(* POU _FB_BACnet_AdsConn, ST *)
FUNCTION_BLOCK _FB_BACnet_AdsConn
VAR_INPUT
	bAutoReload			: BOOL := TRUE; (* TRUE --> reload on device operational state and other changes *)
	bReload				: BOOL; (* FALSE --> TRUE refresh information *)
	bIsClient			: BOOL; (* TRUE --> Connection with client device (remote server) *)
END_VAR
VAR_IN_OUT
	bDevOperational		: BOOL;
	sAmsNetId			: T_AmsNetId;
	tDevObjId			: T_BACnet_ObjectIdentifier;
END_VAR
VAR_OUTPUT
	bReady				: BOOL;
	bBusy				: BOOL;
	bDone				: BOOL;
	bError				: BOOL;
	nErrorId			: UINT;
	stBACnetAds			: ST_BACnet_AdsConnection;
END_VAR
VAR
	_BACnetAmsNetID		: T_AmsNetId;
	_fbAdsRead			: FW_AdsRead;
	_arrAdsBuf			: ARRAY[0..13] OF DWORD;
	_rtrigReload		: R_TRIG;
	_rtrigOP			: R_TRIG;
	_i					: INT;
	_nDevObjects		: UDINT;
	_nObjIdx			: UDINT;
	_nAmsPort			: UINT;
	_tObjId				: T_BACnet_ObjectIdentifier := 16#FFFFFFFF;
END_VAR
(*
#define ADSIGRP_BACNET_CLIENT_COM_PARAMETER                      0x010

typedef struct _BACnetDevComData
{
      BACnetObjectIdentifier deviceObjIdentifier;
      BACnetAddress                  netAddress;                      // 10 Byte
      WORD                                 UdpPort;
      DWORD                                IPadress;       
      WORD                                 maxApdu;                         // wird im "Iam" Frame gesetzt
      WORD                                 vendorId;                        // wird im "Iam" Frame gesetzt
      DWORD                                maxSegments;                     // 0 == unspecified number of segments
      DWORD                                segmentTimeout;            // wenn 0 dann Defaultwerte des Devices nehmen 
      DWORD                                apduTimeout;                     // wenn 0 dann Defaultwerte des Devices nehmen
      DWORD                                nApduRetries;              // wenn 0 dann Defaultwerte des Devices nehmen
      BYTE                                 ethernetMacAddr[6];   // Ethernet MAC Address
      BYTE                                 segmentsSupported;         // segmentation both, transmit, receive, no (0 == segmentation both)
      BYTE                                 reserved;
} BACnetDevComData, *PBACnetDevComData;

-----------------------------------------------------
Server:

AdsReadInd, IndexGroup:
#define ADSIGRP_BACNET_GET_OBJECT_LIST                                 0x009

indexOffset == 0 -> Anzahl der Objekte

gerader Index -> Objekttyp
ungerader Index -> ObjetInstanz

IndexOffset 2 sollte daher die DeviceID des Servers sein
*)

(* ads communication *)
_fbAdsRead(
	sNetId		:= _BACnetAmsNetID,
	nPort		:= ,
	nIdxGrp		:= ,
	nIdxOffs	:= ,
	cbReadLen	:= SIZEOF(_arrAdsBuf),
	pReadBuff	:= ADR(_arrAdsBuf),
	bExecute	:= ,
	tTimeout	:= BACnet_ADSTimeOut,
	bBusy		=> ,
	bError		=> ,
	nErrId		=> ,
	cbRead		=> );

(* catch reload event trigger *)
_rtrigReload(CLK:= bReload, Q=> );
_rtrigOP(CLK:= bDevOperational, Q=> );

(* state machine *)
CASE _i OF

	0: (* Idle *)
		IF sAmsNetId = '' THEN
			(* NetId not OK, return with error *)
			nErrorId := BACnet_ERR_ADS_NO_VALID_NET_ID;
			stBACnetAds.bValid := FALSE;
			_BACnetAmsNetID := '';
		ELSIF (F_BACnet_GetObjType(tDevObjId) <> BACnetObjectType_Device) THEN
			(* Object type is not device *)
			nErrorId := BACnet_ERR_ADS_ObjectId;
			stBACnetAds.bValid := FALSE;
			_tObjId := 0;
		ELSIF	_rtrigReload.Q
			OR	(		(		(sAmsNetId <> stBACnetAds.sAmsNetId)
							OR	(tDevObjId <> _tObjId)
							OR	(_BACnetAmsNetID <> sAmsNetId)
							OR	_rtrigOP.Q
						)
					AND	bAutoReload
				)
		THEN
			IF (NOT bDevOperational) THEN
				(* BACnet adapter error *)
				nErrorId := BACnet_ERR_ADS_DeviceOP;
				stBACnetAds.bValid := FALSE;
			ELSE
				nErrorId := BACnet_ERR_NO_ERROR;
				_i := 1;
				(* store connection info *)
				_BACnetAmsNetID	:= sAmsNetId;
				_tObjId := tDevObjId;
			END_IF
		END_IF
		bDone := FALSE;

	(* Determin the AMS port *)
	1:
		IF _fbAdsRead.bExecute THEN
			IF _fbAdsRead.bError THEN
				IF ((UDINT_TO_DWORD(_fbAdsRead.nErrId) AND 16#0000FFFF) = 16#0703) THEN
					(* couldn't read service for AMS port of the device - maybe R6 stack running *)
					nErrorId := BACnet_ERR_ADS_LegacyStack;
				ELSE
					nErrorId := BACnet_ERR_ADS_Read;
				END_IF
				_fbAdsRead.bExecute := FALSE;
				_i := 100;
				stBACnetAds.bValid := FALSE;
			ELSIF (NOT _fbAdsRead.bBusy) THEN
				_fbAdsRead.bExecute := FALSE;
				(* check if port info is valid *)
				IF (_fbAdsRead.cbRead = 2) THEN
					_nAmsPort := DWORD_TO_UINT(_arrAdsBuf[0] AND 16#0000FFFF);
					(* length ok? *)
					IF _nAmsPort >= 1000 THEN
						IF bIsClient THEN
							_i := 100;
							stBACnetAds.nDeviceId := F_BACnet_GetObjInstance(tDevObjId);
						ELSE
							_i := 11;
						END_IF
					ELSE
						(* wrong length, abort *)
						_i := 100;
						nErrorId := BACnet_ERR_ADS_AmsPort;
						stBACnetAds.bValid := FALSE;
					END_IF
				ELSE
					nErrorId := BACnet_ERR_ADS_Data;
					_i := 100;
					stBACnetAds.bValid := FALSE;
				END_IF
			END_IF
		ELSE
			(* start ADS reading *)
			_fbAdsRead.bExecute := TRUE;
			_fbAdsRead.nIdxGrp := BACnet_ADSIGRP_DEV_R_GETADSPORTBYDEVID;
			_fbAdsRead.nPort := 65535;
			_fbAdsRead.nIdxOffs := tDevObjId;
		END_IF

	(* try READ server info -object list length- *)
	11:
		IF _fbAdsRead.bExecute THEN
			IF _fbAdsRead.bError THEN
				_fbAdsRead.bExecute := FALSE;
				_i := 100;
				nErrorId := BACnet_ERR_ADS_Read;
				stBACnetAds.bValid := FALSE;
			ELSIF (NOT _fbAdsRead.bBusy) THEN
				_fbAdsRead.bExecute := FALSE;
				(* check if object list is valid *)
				IF (_fbAdsRead.cbRead = 4) THEN
					_nDevObjects := _arrAdsBuf[0];
					(* length ok? *)
					IF _nDevObjects >= 1 THEN
						_i := 12;
						_nObjIdx := 0;
					ELSE
						(* wrong length, abort *)
						_i := 100;
						nErrorId := BACnet_ERR_ADS_ObjListEmpty;
						stBACnetAds.bValid := FALSE;
					END_IF
				ELSE
					nErrorId := BACnet_ERR_ADS_Data;
					_i := 100;
					stBACnetAds.bValid := FALSE;
				END_IF
			END_IF
		ELSE
			(* start ADS reading *)
			_fbAdsRead.bExecute := TRUE;
			_fbAdsRead.nIdxGrp := BACnet_ADSIGRP_GET_OBJECT_LIST;
			_fbAdsRead.nPort := _nAmsPort;
			_fbAdsRead.nIdxOffs := 0;
		END_IF

	(* try READ server info -object type- *)
	12:
		IF _fbAdsRead.bExecute THEN
			IF _fbAdsRead.bError THEN
				_fbAdsRead.bExecute := FALSE;
				_i := 100;
				nErrorId := BACnet_ERR_ADS_Read;
				stBACnetAds.bValid := FALSE;
			ELSIF (NOT _fbAdsRead.bBusy) THEN
				_fbAdsRead.bExecute := FALSE;
				(* check if type is valid *)
				IF (_fbAdsRead.cbRead = 4) THEN
					IF (_arrAdsBuf[0] = BACnetObjectType_Device) THEN
						(* device object found, go on *)
						_i := 13;
					ELSE
						(* wrong object type, next list entry *)
						_i := 12; (* remain in current step *)
						_nObjIdx := _nObjIdx + 1;
					END_IF
				ELSE
					nErrorId := BACnet_ERR_ADS_Data;
					_i := 100;
					stBACnetAds.bValid := FALSE;
				END_IF
			END_IF
		ELSE
			(* start ADS reading *)
			IF _nObjIdx < _nDevObjects THEN
				_fbAdsRead.bExecute := TRUE;
				_fbAdsRead.nIdxGrp := BACnet_ADSIGRP_GET_OBJECT_LIST;
				_fbAdsRead.nIdxOffs := (_nObjIdx * 2) + 2;
				_fbAdsRead.nPort := _nAmsPort;
			ELSE
				(* no device found, abort *)
				nErrorId := BACnet_ERR_ADS_NoDevice;
				_i := 100;
				stBACnetAds.bValid := FALSE;
			END_IF
		END_IF

	(* try READ server info -object instance- *)
	13:
		IF _fbAdsRead.bExecute THEN
			IF _fbAdsRead.bError THEN
				_fbAdsRead.bExecute := FALSE;
				_i := 100;
				nErrorId := BACnet_ERR_ADS_Read;
				stBACnetAds.bValid := FALSE;
			ELSIF (NOT _fbAdsRead.bBusy) THEN
				_fbAdsRead.bExecute := FALSE;
				(* preset done *)
				_i := 100;
				(* check if ID is valid *)
				IF (_fbAdsRead.cbRead = 4) THEN
					IF (_arrAdsBuf[0] <= 16#3FFFFF) THEN
						IF (F_BACnet_GetObjInstance(tDevObjId) = _arrAdsBuf[0]) THEN
							stBACnetAds.nDeviceId := F_BACnet_GetObjInstance(tDevObjId);
						ELSE
							nErrorId := BACnet_ERR_ADS_ObjIdMissmatch;
							stBACnetAds.bValid := FALSE;
						END_IF
					ELSE
						nErrorId := BACnet_ERR_ADS_ObjInstance;
						stBACnetAds.bValid := FALSE;
					END_IF
				ELSE
					nErrorId := BACnet_ERR_ADS_Data;
					stBACnetAds.bValid := FALSE;
				END_IF
			END_IF
		ELSE
			(* start ADS reading *)
			_fbAdsRead.bExecute := TRUE;
			_fbAdsRead.nIdxGrp := BACnet_ADSIGRP_GET_OBJECT_LIST;
			_fbAdsRead.nIdxOffs := (_nObjIdx * 2) + 1;
			_fbAdsRead.nPort := _nAmsPort;
		END_IF

	100: (* Done *)
		bDone := (nErrorId = BACnet_ERR_NO_ERROR);
		IF (NOT bDone) THEN
			stBACnetAds.bValid := FALSE;
		ELSE
			(* set states *)
			stBACnetAds.bServer := (NOT bIsClient);
			stBACnetAds.bClient := bIsClient;
			stBACnetAds.bValid := TRUE;
			(* count update *)
			stBACnetAds.nReload := stBACnetAds.nReload + 1;
		END_IF
		(* remind device AmsNetID and port *)
		stBACnetAds.sAmsNetId	:= _BACnetAmsNetID;
		stBACnetAds.nAmsPort	:= _nAmsPort;
		(* go idle *)
		_i := 0;

END_CASE

(* set error flag *)
bError	:= (nErrorId <> BACnet_ERR_NO_ERROR);
bBusy	:= _i > 0;
bReady	:= (NOT bError) AND ((NOT bBusy) OR bReady);
END_FUNCTION_BLOCK

(* POU F_BACnet_GetObjType, ST *)
FUNCTION F_BACnet_GetObjType : E_BACNETOBJECTTYPE
VAR_INPUT
	nObjectId : DWORD;
END_VAR
VAR
END_VAR
F_BACnet_GetObjType := DWORD_TO_WORD(SHR((nObjectId AND 16#FFC00000), 22));
END_FUNCTION

(* POU F_BACnet_GetObjInstance, ST *)
FUNCTION F_BACnet_GetObjInstance : UDINT
VAR_INPUT
	nObjectId : DWORD;
END_VAR
VAR
END_VAR
F_BACnet_GetObjInstance := nObjectId AND 16#003FFFFF;
END_FUNCTION

(* POU _FB_BACnet_PidTune, ST *)
FUNCTION_BLOCK _FB_BACnet_PidTune
VAR_INPUT
	bStart	: BOOL;
	bStop	: BOOL; (* Abort tuning process *)
	fSetY	: REAL;
	fX		: REAL;
	fDeadband	: REAL;
	tTimeout: TIME := T#15m;
	fMinY	: REAL;
	fMaxY	: REAL;
	fCycleTime : REAL; (* cycle time in seconds [s]; 0 = use internal measuring *)
	eMode	: E_BACNETPIDTUNINGMODE := BACnetPIDTuningMode_PI;
END_VAR
VAR_IN_OUT
	fY		: REAL;
END_VAR
VAR_OUTPUT
	fPID_Kp	: REAL;
	fPID_Ki	: REAL;
	fPID_Kd	: REAL;
	eAction	: E_BACNETACTION;
	bSetY	: BOOL;
	bWaitY	: BOOL;
	bWaitX	: BOOL;
	bReady	: BOOL;
	bBusy	: BOOL;
	bDone	: BOOL;
	bAborted: BOOL;
	bTimeout: BOOL;
END_VAR
VAR
	_oldY	: REAL;
	_fbPT1_D: FB_BACnet_PT1;
	_step : INT;
	_sysTime	: GETCPUCOUNTER;
	_Time : T_LARGE_INTEGER;
	_TimeOld : T_LARGE_INTEGER;
	_TimeStart : T_LARGE_INTEGER;
	_fbAvg : FB_BACnet_AvgValue;
	_fCycleTime : REAL;
	_oldX : REAL;
	_highest : ARRAY[0..9] OF ARRAY[0..1] OF REAL;
	_HighestPoint : ARRAY[0..1] OF REAL;
	_nFifoHigh : INT;
	_nFifoCount : DINT;
	_fDsum : REAL;
	_fDhigh : REAL;
	_tonTimeout : TON;
	_tofYRemain : TOF;
	_tofXRemain : TOF;
	_StartPoint : ARRAY[0..1] OF REAL;
	_EndPoint : ARRAY[0..1] OF REAL;
	_fn : REAL;
	_fTu : REAL;
	_fPID_Tn : REAL;
	_fPID_Tv : REAL;
	_tonStartDelay : TON;
	_fStartX : REAL;
	_fStartY : REAL;
	_tonMeasureTrigger : TON;
	_Xp : REAL;
	_D	: REAL;
	_bDsink : BOOL;
	_bMinScanTime : BOOL;
END_VAR
_tofYRemain(IN:= (fY <> _oldY), PT:= (tTimeout / 100), Q=> , ET=> );
_tofXRemain(IN:= (ABS(_fbPT1_D.Y) > ABS(fDeadband)), PT:= (tTimeout / 100), Q=> , ET=> );

(* timeout *)
_tonTimeout(IN:= , PT:= tTimeout, Q=> , ET=> );

(* record exact cycle time *)
_TimeOld := _Time;
_sysTime(
	cpuCntLoDW=> _Time.dwLowPart,
	cpuCntHiDW=> _Time.dwHighPart);

(* average filter for input value *)
_fbAvg(X:= fX, n:= 100, Y=> );
(* trigger timer *)
_tonMeasureTrigger(IN:= NOT _tonMeasureTrigger.Q, PT:= (tTimeout / 300), Q=> , ET=> );
(* calculate gradient on trigger event *)
IF _tonMeasureTrigger.Q THEN
	_fCycleTime := _F_BACnet_SysTimeDiff(_Time, _TimeOld); (* [s] *)
	IF (_fCycleTime > 0.0) THEN
		(* calculate gradient *)
		_D := (_fbAvg.Y - _oldX) / _fCycleTime;
	END_IF
	(* reset average filter *)
	_fbAvg(X:= _fbAvg.Y, n:= 0, Y=> );
	(* reset trigger *)
	_tonMeasureTrigger(IN := FALSE);
END_IF
(* gradient filter *)
_fbPT1_D(X:= _D, T:= TIME_TO_REAL(tTimeout) / 1000.0 / 200.0, Tcycle:= fCycleTime, Y=> );

bWaitX := _tofXRemain.Q AND (_step = 0);
bWaitY := _tofYRemain.Q AND (_step = 0);
bReady :=	(NOT bWaitX)
		AND	(NOT bWaitY)
		AND (_step = 0);
_tonStartDelay(IN:= bStart AND bReady, PT:= (tTimeout / 100), Q=> , ET=> );

bSetY := FALSE;

CASE _step OF

	0:
		IF bStart AND (NOT bStop) THEN
			IF _tonStartDelay.Q THEN
				bReady := FALSE;
				_StartPoint[0] := 0.0;
				_StartPoint[1] := fX;
				_step := 10;
				_TimeStart := _Time;
				_fStartY := fY;
				_fStartX := fX;
				_tonTimeout.IN := FALSE;
			ELSE
				_tonTimeout.IN := TRUE;
			END_IF
		ELSE
			bWaitY := FALSE;
			bWaitX := FALSE;
			_tonTimeout.IN := FALSE;
		END_IF

	10: (* wait start condition *)
		fY := fSetY;
		bWaitX := TRUE;
		bSetY := TRUE;
		_tonTimeout.IN := TRUE;
		IF bStop THEN
			_step := 200;
		ELSIF (_tonTimeout.Q) THEN
			_step := 200;
		ELSIF	(_fbAvg.Y > _fStartX + ABS(fDeadband))
			OR	(_fbAvg.Y < _fStartX - ABS(fDeadband))
		THEN
			_step := 20;
			_nFifoHigh := 0;
			_fDhigh := 0.0;
			_nFifoCount := 0;
			_fDsum := 0.0;
			_tonTimeout.IN := FALSE;
		END_IF

	20: (* record *)
		bWaitX := TRUE;
		bSetY := TRUE;
		_tonTimeout.IN := TRUE;
		IF bStop THEN
			_step := 200;
		ELSIF _tonTimeout.Q THEN
			_step := 200;
			bTimeout := TRUE;
		ELSIF	((_D > _fDhigh) AND (_fbAvg.Y > _fStartX)) (* direct system / pos. acceleration *)
			OR	((_D < _fDhigh) AND (_fbAvg.Y < _fStartX)) (* reverse system / neg. acceleration *)
		THEN
			_fDsum := _fDsum + _fbPT1_D.Y;
			IF (_nFifoCount >= 10) THEN
				_fDsum := _fDsum - _highest[_nFifoHigh][1];
			END_IF
			(* remind highest gradiant *)
			_fDhigh := _D;
			(* fill into FIFO *)
			_highest[_nFifoHigh][0] := _F_BACnet_SysTimeDiff(_Time, _TimeStart);
			_highest[_nFifoHigh][1] := _fbPT1_D.Y;
			(* remind highest point *)
			_HighestPoint[0] := _highest[_nFifoHigh][0];	(* t [s] *)
			_HighestPoint[1] := _fbAvg.Y;							(* X [1] *)
			(* count FIFO position and counter *)
			_nFifoHigh := (_nFifoHigh + 1) MOD 10;
			_nFifoCount := _nFifoCount + 1;
		END_IF
		(* check scan time *)
		_bMinScanTime := (_F_BACnet_SysTimeDiff(_Time, _TimeStart) >= ((TIME_TO_REAL(tTimeout) / 1000.0) / 10.0));
		(* exit, when acceleration sinks *)
		IF		(_nFifoCount >= 10)
			AND	_bMinScanTime
		THEN
			(* sink detected, when gradient fells beneath 30% of averaged gradient *)
			_bDsink := (ABS(_fbPT1_D.Y) <= (ABS(_fDsum / 10.0) * 0.3));
		ELSE
			_bDsink := FALSE;
		END_IF
		IF 		_bDsink
			OR	(		_bMinScanTime
					AND	(ABS(_fbPT1_D.Y) < (ABS(_fDhigh) * 0.1)) (* less 10% of max. gradient *)
					AND	(_nFifoCount > 1)
				)
		THEN
			_step := 90;
			_EndPoint[0] := _F_BACnet_SysTimeDiff(_Time, _TimeStart);
			_EndPoint[1] := fX;
			_tonTimeout.IN := FALSE;
		END_IF

	90:
		_step := 100;
		fY := _fStartY;

		IF (_fDhigh <> 0.0) AND (fSetY - _fStartY <> 0.0) THEN
			(* calculate linear function offset *)
			_fn := _HighestPoint[1] - (_fDhigh * _HighestPoint[0]);

			(* calculate X intersection with minimum value (Tu)
				Tu = (Ymin - N) / D			 	*)
			_fTu := ABS((_StartPoint[1] - _fn) / _fDhigh);

			IF (_fTu > 0.0) THEN
				(* calculate Kp *)
				_Xp := _fDhigh * _fTu * (fMaxY - fMinY) / (fSetY - _fStartY);
				IF (_Xp >= 0.0) THEN
					eAction := BACnetAction_direct;
				ELSE
					eAction := BACnetAction_reverse;
				END_IF
				_Xp := ABS(_Xp);

				(* decide between tuning modes *)
				CASE eMode OF
					BACnetPIDTuningMode_P:
						(* calculate P controller *)
						_fPID_Tn := 0.0;
						_fPID_Tv := 0.0;
						fPID_Kp := _Xp;
						fPID_Ki := 0.0;
						fPID_Kd := 0.0;

					BACnetPIDTuningMode_PI:
						(* calculate PI controller *)
						_fPID_Tn := 3.3 * _fTu;
						_fPID_Tv := 0.0;
						fPID_Kp := 1.2 * _Xp;
						fPID_Ki := (1 / _fPID_Tn) * fPID_Kp;
						fPID_Kd := 0.0;

					BACnetPIDTuningMode_PD:
						(* calculate PI controller *)
						_fPID_Tn := 0.0;
						_fPID_Tv := 0.25 * _fTu;
						fPID_Kp := 0.83 * _Xp;
						fPID_Ki := 0.0;
						fPID_Kd := _fPID_Tv * fPID_Kp;

					BACnetPIDTuningMode_PID:
						(* calculate PID controller *)
						_fPID_Tn := 2.0 * _fTu;
						_fPID_Tv := 0.5 * _fTu;
						fPID_Kp := 0.83 * _Xp;
						IF (_fPID_Tn <> 0.0) THEN
							fPID_Ki := (1 / _fPID_Tn) * fPID_Kp;
						ELSE
							fPID_Ki := 0.0;
						END_IF
						fPID_Kd := _fPID_Tv * fPID_Kp;

				END_CASE
			ELSE
				_step := 200;
			END_IF
		ELSE
			_step := 200;
		END_IF


	100:
		IF (NOT bStart) THEN
			_step := 0;
		END_IF

	200:
		fY := _fStartY;
		_tonTimeout.IN := FALSE;
		IF (NOT bStart) THEN
			_step := 0;
			bTimeout := FALSE;
		END_IF

END_CASE

bAborted := _step = 200;
bDone := _step = 100;
bBusy := _step > 0 AND (NOT bDone) AND (NOT bAborted);

_oldY := fY;
_oldX := _fbAvg.Y;
END_FUNCTION_BLOCK

(* POU FB_BACnet_PT1, ST *)
FUNCTION_BLOCK FB_BACnet_PT1
VAR_INPUT
	X : REAL; (* input value *)
	T : REAL; (* damping time [s] *)
	Tcycle : REAL; (* cycle time [s] of task; 0 = use internal measuring *)
END_VAR
VAR_OUTPUT
	Y : REAL; (* damped value *)
END_VAR
VAR
	_sysTime	: GETCPUCOUNTER;
	_Time		: T_LARGE_INTEGER;
	_TimeOld	: T_LARGE_INTEGER;
	_cycleTime	: REAL;
	_Yold : REAL;
	_FirstScan : BOOL := TRUE;
END_VAR
(* determine cycle time *)
IF Tcycle = 0.0 THEN
	_TimeOld := _Time;
	_sysTime(cpuCntLoDW=> _Time.dwLowPart, cpuCntHiDW=> _Time.dwHighPart);
	_cycleTime := _F_BACnet_SysTimeDiff(In1:=_Time, In2:=_TimeOld);
ELSE
	_cycleTime := Tcycle;
END_IF

(* exit on wrong cycle time *)
IF _cycleTime <= 0.0 THEN
	RETURN;
END_IF

(* initialize and check on zero/negative damping time *)
IF (T <= 0.0) OR _FirstScan THEN
	Y := X;
	_Yold := Y;
	_FirstScan := FALSE;
	RETURN;
END_IF

(* remind last result *)
_Yold := Y;

(* calculate result *)
Y := 1 / ((T / _cycleTime) + 1) * (X - _Yold) + _Yold;
END_FUNCTION_BLOCK

(* POU FB_BACnet_AvgValue, ST *)
FUNCTION_BLOCK FB_BACnet_AvgValue
VAR_INPUT
	X	: REAL; (* input value to average *)
	n	: INT; (* number of averages (0 = no average --> Y = X) *)
END_VAR
VAR_OUTPUT
	Y	: REAL; (* average result *)
END_VAR
VAR
	_n	: INT := 0;
	_Xn : LREAL;
END_VAR
IF (_n > n) THEN
	_n := n;
END_IF
IF (_n = 0) OR (n = 0) THEN
	_Xn := REAL_TO_LREAL(X);
ELSE
	_Xn := ((_Xn * _n) + REAL_TO_LREAL(X)) / INT_TO_LREAL(_n + 1);
END_IF
_n := _n + 1;
Y := LREAL_TO_REAL(_Xn);
END_FUNCTION_BLOCK

(* POU F_BACnet_AnalogPV, ST *)
FUNCTION F_BACnet_AnalogPV : REAL
VAR_INPUT
	bEnable	: BOOL; (* TRUE = commit to stack, FALSE = do-nothing *)
	bNull	: BOOL; (* TRUE = clear priority, FALSE = write value from input *)
	rValue	: REAL;
END_VAR
IF (bEnable) THEN
	IF (bNull) THEN
		F_BACnet_AnalogPV := F_BACnet_RealNull();
	ELSE
		F_BACnet_AnalogPV := rValue;
	END_IF
ELSE
	F_BACnet_AnalogPV := F_BACnet_NAN();
END_IF
END_FUNCTION

(* POU F_BACnet_RealNull, ST *)
FUNCTION F_BACnet_RealNull : DWORD
(* function that generates <not-a-number> real state *)
F_BACnet_RealNull:=16#7FFF0000;
END_FUNCTION

(* POU F_BACnet_NAN, ST *)
FUNCTION F_BACnet_NAN : REAL
(* function that generates <not-a-number> real state *)
VAR_INPUT
END_VAR
VAR
	res : POINTER TO DWORD;
END_VAR
res:=ADR(F_BACnet_NAN);
res^:=16#7FFFFFFF;
END_FUNCTION

(* POU F_BACnet_CheckDay, ST *)
FUNCTION F_BACnet_CheckDay : USINT
VAR_IN_OUT
	nIn	: BYTE;
END_VAR
VAR
END_VAR
IF nIn > 32 OR nIn = 0 THEN
	F_BACnet_CheckDay := 255;
ELSE
	F_BACnet_CheckDay := nIn;
END_IF
nIn := F_BACnet_CheckDay;
END_FUNCTION

(* POU F_BACnet_CheckDayOfWeek, ST *)
FUNCTION F_BACnet_CheckDayOfWeek : USINT
VAR_IN_OUT
	nIn	: BYTE;
END_VAR
VAR
END_VAR
IF nIn > 7 OR nIn = 0 THEN
	F_BACnet_CheckDayOfWeek := 255;
ELSE
	F_BACnet_CheckDayOfWeek := nIn;
END_IF
nIn := F_BACnet_CheckDayOfWeek;
END_FUNCTION

(* POU F_BACnet_CheckHour, ST *)
FUNCTION F_BACnet_CheckHour : USINT
VAR_IN_OUT
	nIn	: BYTE;
END_VAR
VAR
END_VAR
IF nIn > 23 THEN
	F_BACnet_CheckHour := 255;
ELSE
	F_BACnet_CheckHour := nIn;
END_IF
nIn := F_BACnet_CheckHour;
END_FUNCTION

(* POU F_BACnet_CheckHundredths, ST *)
FUNCTION F_BACnet_CheckHundredths : USINT
VAR_IN_OUT
	nIn	: BYTE;
END_VAR
VAR
END_VAR
IF nIn > 99 THEN
	F_BACnet_CheckHundredths := 255;
ELSE
	F_BACnet_CheckHundredths := nIn;
END_IF
nIn := F_BACnet_CheckHundredths;
END_FUNCTION

(* POU F_BACnet_CheckMinute, ST *)
FUNCTION F_BACnet_CheckMinute : USINT
VAR_IN_OUT
	nIn	: BYTE;
END_VAR
VAR
END_VAR
IF nIn > 59 THEN
	F_BACnet_CheckMinute := 255;
ELSE
	F_BACnet_CheckMinute := nIn;
END_IF
nIn := F_BACnet_CheckMinute;
END_FUNCTION

(* POU F_BACnet_CheckMonth, ST *)
FUNCTION F_BACnet_CheckMonth : USINT
VAR_IN_OUT
	nIn	: BYTE;
END_VAR
VAR
END_VAR
IF nIn > 14 OR nIn = 0 THEN
	F_BACnet_CheckMonth := 255;
ELSE
	F_BACnet_CheckMonth := nIn;
END_IF
nIn := F_BACnet_CheckMonth;
END_FUNCTION

(* POU F_BACnet_CheckSecond, ST *)
FUNCTION F_BACnet_CheckSecond : USINT
VAR_IN_OUT
	nIn	: BYTE;
END_VAR
VAR
END_VAR
IF nIn > 59 THEN
	F_BACnet_CheckSecond := 255;
ELSE
	F_BACnet_CheckSecond := nIn;
END_IF
nIn := F_BACnet_CheckSecond;
END_FUNCTION

(* POU F_BACnet_CheckWeekOfMonth, ST *)
FUNCTION F_BACnet_CheckWeekOfMonth : USINT
VAR_IN_OUT
	nIn	: BYTE;
END_VAR
VAR
END_VAR
IF nIn > 7 OR nIn = 0 THEN
	F_BACnet_CheckWeekOfMonth := 255;
ELSE
	F_BACnet_CheckWeekOfMonth := nIn;
END_IF
nIn := F_BACnet_CheckWeekOfMonth;
END_FUNCTION

(* POU F_BACnet_CheckYear, ST *)
FUNCTION F_BACnet_CheckYear : USINT
VAR_IN_OUT
	nIn	: BYTE;
END_VAR
VAR
END_VAR
F_BACnet_CheckYear := nIn;
nIn := F_BACnet_CheckYear;
END_FUNCTION

(* POU F_BACnet_DateHasPlaceholder, ST *)
FUNCTION F_BACnet_DateHasPlaceholder : BOOL
VAR_INPUT
	stDate		: ST_BACnet_Date;
END_VAR
F_BACnet_DateHasPlaceholder := (stDate.nDay = 16#FF) OR (stDate.nDayOfWeek = 16#FF) OR (stDate.nMonth = 16#FF) OR (stDate.nYear = 16#FF);
END_FUNCTION

(* POU F_BACnet_DateMerge, ST *)
FUNCTION F_BACnet_DateMerge : ST_BACnet_Date (* This function replacing placeholders in both dates and returning the result (if no placeholder is given, date1 will be prefered) *)
VAR_INPUT
	stDate1		: ST_BACnet_Date;
	stDate2		: ST_BACnet_Date;
END_VAR
VAR
END_VAR
IF stDate1.nDay = 16#FF THEN
	F_BACnet_DateMerge.nDay := F_BACnet_CheckDay(stDate2.nDay);
ELSE
	F_BACnet_DateMerge.nDay := F_BACnet_CheckDay(stDate1.nDay);
END_IF
IF stDate1.nDayOfWeek = 16#FF THEN
	F_BACnet_DateMerge.nDayOfWeek := F_BACnet_CheckDayOfWeek(stDate2.nDayOfWeek);
ELSE
	F_BACnet_DateMerge.nDayOfWeek := F_BACnet_CheckDayOfWeek(stDate1.nDayOfWeek);
END_IF
IF stDate1.nMonth = 16#FF THEN
	F_BACnet_DateMerge.nMonth := F_BACnet_CheckMonth(stDate2.nMonth);
ELSE
	F_BACnet_DateMerge.nMonth := F_BACnet_CheckMonth(stDate1.nMonth);
END_IF
IF stDate1.nYear = 16#FF THEN
	F_BACnet_DateMerge.nYear := F_BACnet_CheckYear(stDate2.nYear);
ELSE
	F_BACnet_DateMerge.nYear := F_BACnet_CheckYear(stDate1.nYear);
END_IF
END_FUNCTION

(* POU F_BACnet_DateTime_TO_TimeStruct, ST *)
FUNCTION F_BACnet_DateTime_TO_TimeStruct : TIMESTRUCT
VAR_INPUT
	IN	: ST_BACnet_DateTime;
END_VAR
F_BACnet_DateTime_TO_TimeStruct.wDay			:= BYTE_TO_WORD(IN.stDate.nDay);
F_BACnet_DateTime_TO_TimeStruct.wDayOfWeek		:= BYTE_TO_WORD(IN.stDate.nDayOfWeek MOD 7);
F_BACnet_DateTime_TO_TimeStruct.wDay			:= BYTE_TO_WORD(IN.stDate.nDay);
F_BACnet_DateTime_TO_TimeStruct.wMonth			:= BYTE_TO_WORD(IN.stDate.nMonth);
F_BACnet_DateTime_TO_TimeStruct.wYear			:= BYTE_TO_WORD(IN.stDate.nYear) + 1900;
F_BACnet_DateTime_TO_TimeStruct.wHour			:= BYTE_TO_WORD(IN.stTime.nHour);
F_BACnet_DateTime_TO_TimeStruct.wMinute			:= BYTE_TO_WORD(IN.stTime.nMinute);
F_BACnet_DateTime_TO_TimeStruct.wSecond			:= BYTE_TO_WORD(IN.stTime.nSecond);
F_BACnet_DateTime_TO_TimeStruct.wMilliseconds	:= BYTE_TO_WORD(IN.stTime.nHundredths) * 10;
END_FUNCTION

(* POU F_BACnet_DateTimeString, ST *)
FUNCTION F_BACnet_DateTimeString : STRING(19)
VAR_IN_OUT
	stDateTime		: ST_BACnet_DateTime;
END_VAR
VAR
	str : STRING;
END_VAR
str := '';
IF stDateTime.stDate.nDay >= 1 THEN
	IF stDateTime.stDate.nDay <= 9 THEN
		str := CONCAT(str, CONCAT('0', BYTE_TO_STRING(stDateTime.stDate.nDay)));
	ELSIF stDateTime.stDate.nDay <= 31 THEN
		str := CONCAT(str, BYTE_TO_STRING(stDateTime.stDate.nDay));
	ELSE
		str := CONCAT(str, '**');
	END_IF
ELSE
	str := CONCAT(str, '**');
END_IF

str := CONCAT(str, '.');
IF stDateTime.stDate.nMonth >= 1 THEN
	IF stDateTime.stDate.nMonth <= 9 THEN
		str := CONCAT(str, CONCAT('0', BYTE_TO_STRING(stDateTime.stDate.nMonth)));
	ELSIF stDateTime.stDate.nMonth <= 12 THEN
		str := CONCAT(str, BYTE_TO_STRING(stDateTime.stDate.nMonth));
	ELSE
		str := CONCAT(str, '**');
	END_IF
ELSE
	str := CONCAT(str, '**');
END_IF

str := CONCAT(str, '.');
IF stDateTime.stDate.nYear < 16#FF THEN
	str := CONCAT(str, UINT_TO_STRING(BYTE_TO_UINT(stDateTime.stDate.nYear) + 1900));
ELSE
	str := CONCAT(str, '****');
END_IF

str := CONCAT(str, ' ');
str := CONCAT(str, F_BACnet_TimeString(stDateTime.stTime));
F_BACnet_DateTimeString := str;
END_FUNCTION

(* POU F_BACnet_TimeString, ST *)
FUNCTION F_BACnet_TimeString : STRING(12)
VAR_IN_OUT
	stTime : ST_BACnet_Time;
END_VAR
VAR
	str : STRING;
END_VAR
str := '';
IF stTime.nHour <= 9 THEN
	str := CONCAT(str, CONCAT('0', BYTE_TO_STRING(stTime.nHour)));
ELSIF stTime.nHour <= 23 THEN
	str := CONCAT(str, BYTE_TO_STRING(stTime.nHour));
ELSE
	str := CONCAT(str, '**');
END_IF

str := CONCAT(str, ':');
IF stTime.nMinute <= 9 THEN
	str := CONCAT(str, CONCAT('0', BYTE_TO_STRING(stTime.nMinute)));
ELSIF stTime.nMinute <= 59 THEN
	str := CONCAT(str, BYTE_TO_STRING(stTime.nMinute));
ELSE
	str := CONCAT(str, '**');
END_IF

str := CONCAT(str, ':');
IF stTime.nSecond <= 9 THEN
	str := CONCAT(str, CONCAT('0', BYTE_TO_STRING(stTime.nSecond)));
ELSIF stTime.nSecond <= 59 THEN
	str := CONCAT(str, BYTE_TO_STRING(stTime.nSecond));
ELSE
	str := CONCAT(str, '**');
END_IF

str := CONCAT(str, '.');
IF stTime.nHundredths <= 9 THEN
	str := CONCAT(str, CONCAT('0', BYTE_TO_STRING(stTime.nHundredths)));
ELSIF stTime.nHundredths <= 99 THEN
	str := CONCAT(str, BYTE_TO_STRING(stTime.nHundredths));
ELSE
	str := CONCAT(str, '**');
END_IF
F_BACnet_TimeString := str;
END_FUNCTION

(* POU F_BACnet_DateUnspecified, ST *)
FUNCTION F_BACnet_DateUnspecified : BOOL
VAR_INPUT
	stDate		: ST_BACnet_Date;
END_VAR
F_BACnet_DateUnspecified := (stDate.nDay = 16#FF) AND (stDate.nDayOfWeek = 16#FF) AND (stDate.nMonth = 16#FF) AND (stDate.nYear = 16#FF);
END_FUNCTION

(* POU F_BACnet_DaysInMonth, ST *)
FUNCTION F_BACnet_DaysInMonth : UDINT (* Returns the numbers of days in given month - 16#FFFFFFFF = unspecified *)
VAR_INPUT
	stBACnetDate		: ST_BACnet_Date;
END_VAR
VAR
	isLeapYear			: BOOL;
	nYear				: UDINT;
END_VAR
IF (stBACnetDate.nMonth = 16#FF) OR (stBACnetDate.nYear = 16#FF) THEN
	(* month and/or year is unspecified *)
	F_BACnet_DaysInMonth := 16#FFFFFFFF;
ELSIF	stBACnetDate.nMonth = 1
	OR	stBACnetDate.nMonth = 3
	OR	stBACnetDate.nMonth = 5
	OR	stBACnetDate.nMonth = 7
	OR	stBACnetDate.nMonth = 8
	OR	stBACnetDate.nMonth = 10
	OR	stBACnetDate.nMonth = 12
THEN
	F_BACnet_DaysInMonth := 31;
ELSE
	IF (stBACnetDate.nMonth = 2) THEN
		(* calculate absolute your number *)
		nYear := stBACnetDate.nYear + 1900;
		(* and check if it is a leap year *)
		isLeapYear := (nYear MOD 4 = 0) AND ((nYear MOD 100 <> 0) OR (nYear MOD 400 = 0));
		(* decide february amount of days *)
		IF (isLeapYear) THEN
		  F_BACnet_DaysInMonth := 29;
		ELSE
		  F_BACnet_DaysInMonth := 28;
		END_IF
	ELSE
		F_BACnet_DaysInMonth := 30;
	END_IF
END_IF
END_FUNCTION

(* POU F_BACnet_EventTransitionFlags, ST *)
FUNCTION F_BACnet_EventTransitionFlags : ST_BACnet_EventTransitionBits
VAR_INPUT
	data	: WORD;
END_VAR
VAR
END_VAR
F_BACnet_EventTransitionFlags.to_normal := _F_BACnet_IsBitFieldBitSet( data:=data, Bit:=BACnetEventTransitionBit_to_normal);
F_BACnet_EventTransitionFlags.to_offnormal := _F_BACnet_IsBitFieldBitSet( data:=data, Bit:=BACnetEventTransitionBit_to_offnormal);
F_BACnet_EventTransitionFlags.to_fault := _F_BACnet_IsBitFieldBitSet( data:=data, Bit:=BACnetEventTransitionBit_to_fault);
END_FUNCTION

(* POU F_BACnet_Get100msDate, ST *)
FUNCTION F_BACnet_Get100msDate : UDINT (* Returns date as 100ms value from 1900 (if year and month are specified!) *)
VAR_INPUT
	stBACnetDate		: ST_BACnet_Date;
END_VAR
VAR
	iValue : UDINT;
	i : BYTE;
	stDate : ST_BACnet_Date;
END_VAR
iValue := 0;
IF stBACnetDate.nYear < 16#FF THEN
	iValue := iValue + BYTE_TO_UDINT(stBACnetDate.nYear) * 365 * 24 * 60 * 60 * 10;
	IF stBACnetDate.nDay >= 1 AND stBACnetDate.nDay <= 12 THEN
		stDate := stBACnetDate;
		FOR i := 1 TO stBACnetDate.nMonth-1 DO
			stDate.nMonth := i;
			iValue := iValue + F_BACnet_DaysInMonth(stDate) * 24 * 60 * 60 * 10;
		END_FOR
	END_IF
END_IF
IF stBACnetDate.nDay >= 1 AND stBACnetDate.nDay <= 31 THEN
	iValue := iValue + BYTE_TO_UDINT(stBACnetDate.nDay) * 24 * 60 * 60 * 10;
END_IF
F_BACnet_Get100msDate := iValue;
END_FUNCTION

(* POU F_BACnet_Get100msTime, ST *)
FUNCTION F_BACnet_Get100msTime : UDINT (* Returns time as 100ms value from 00:00:00.0 *)
VAR_INPUT
	stBACnetTime : ST_BACnet_Time;
END_VAR
VAR
	iValue		: UDINT;
END_VAR
iValue := 0;
IF (stBACnetTime.nHour < 16#FF) THEN
	iValue := iValue + BYTE_TO_UDINT(stBACnetTime.nHour) * 60 * 60 * 10;
END_IF
IF (stBACnetTime.nMinute < 16#FF) THEN
	iValue := iValue + BYTE_TO_UDINT(stBACnetTime.nMinute) * 60 * 10;
END_IF
IF (stBACnetTime.nSecond < 16#FF) THEN
	iValue := iValue + BYTE_TO_UDINT(stBACnetTime.nSecond) * 10;
END_IF
IF (stBACnetTime.nHundredths < 16#FF) THEN
	iValue := iValue + BYTE_TO_UDINT(stBACnetTime.nHundredths) / 10;
END_IF
F_BACnet_Get100msTime := iValue;
END_FUNCTION

(* POU F_BACnet_GetEventTransFlagsData, ST *)
FUNCTION F_BACnet_GetEventTransFlagsData : WORD
VAR_INPUT
	Flags	: ST_BACnet_EventTransitionBits;
END_VAR
VAR
END_VAR
F_BACnet_GetEventTransFlagsData := 16#0005;
IF Flags.to_normal THEN
	F_BACnet_GetEventTransFlagsData := DWORD_TO_WORD(_F_BACnet_SetBitFieldBit(ptrData:=ADR(F_BACnet_GetEventTransFlagsData), Bit:=BACnetEventTransitionBit_to_normal));
END_IF
IF Flags.to_offnormal THEN
	F_BACnet_GetEventTransFlagsData := DWORD_TO_WORD(_F_BACnet_SetBitFieldBit(ptrData:=ADR(F_BACnet_GetEventTransFlagsData), Bit:=BACnetEventTransitionBit_to_offnormal));
END_IF
IF Flags.to_fault THEN
	F_BACnet_GetEventTransFlagsData := DWORD_TO_WORD(_F_BACnet_SetBitFieldBit(ptrData:=ADR(F_BACnet_GetEventTransFlagsData), Bit:=BACnetEventTransitionBit_to_fault));
END_IF
END_FUNCTION

(* POU F_BACnet_GetLimitEnFlagsData, ST *)
FUNCTION F_BACnet_GetLimitEnFlagsData : WORD
VAR_INPUT
	Flags	: ST_BACnet_LimitEnable;
END_VAR
VAR
END_VAR
F_BACnet_GetLimitEnFlagsData := 16#0006;
IF Flags.highLimitEnable THEN
	F_BACnet_GetLimitEnFlagsData := DWORD_TO_WORD(_F_BACnet_SetBitFieldBit(ptrData:=ADR(F_BACnet_GetLimitEnFlagsData), Bit:=BACnetLimitEnableBits_highLimit));
END_IF
IF Flags.lowLimitEnable THEN
	F_BACnet_GetLimitEnFlagsData := DWORD_TO_WORD(_F_BACnet_SetBitFieldBit(ptrData:=ADR(F_BACnet_GetLimitEnFlagsData), Bit:=BACnetLimitEnableBits_lowLimit));
END_IF
END_FUNCTION

(* POU F_BACnet_GetObjectIdString, ST *)
FUNCTION F_BACnet_GetObjectIdString : STRING
VAR_INPUT
	tObjectID : T_BACnet_ObjectIdentifier := 16#FFFFFFFF;
END_VAR
VAR
	nObjType	: UDINT;
	nObjInstance: UDINT;
END_VAR
nObjType	:= F_BACnet_GetObjType(tObjectID);
nObjInstance:= F_BACnet_GetObjInstance(tObjectID);
IF nObjType >= 0 AND nObjType < BACnetObjectType_ZCount THEN
	F_BACnet_GetObjectIdString := CONCAT(CONCAT(arrBACnet_ObjectTypeNameShort[nObjType], ':'), UDINT_TO_STRING(nObjInstance));
ELSE
	F_BACnet_GetObjectIdString := CONCAT('???:', UDINT_TO_STRING(nObjInstance));
END_IF
END_FUNCTION

(* POU F_BACnet_GetObjectListIndex, ST *)
FUNCTION F_BACnet_GetObjectListIndex : DINT
VAR_INPUT
	tObjectId	: T_BACnet_ObjectIdentifier := 16#FFFFFFFF;
END_VAR
VAR_IN_OUT
	stObjIDList	: ST_BACnet_ObjectIdentifierList;
END_VAR
VAR
	iMax : DINT;
	i : DINT;
END_VAR
iMax := stObjIDList.nEntries-1;
F_BACnet_GetObjectListIndex := -1; (* preset: no match *)
FOR i := 0 TO iMax DO
	IF stObjIDList.arrObjList[i] = tObjectId THEN
		F_BACnet_GetObjectListIndex := i; (* match *)
		RETURN;
	END_IF
END_FOR
END_FUNCTION

(* POU F_BACnet_GetObjId, ST *)
FUNCTION F_BACnet_GetObjId : T_BACnet_ObjectIdentifier
VAR_INPUT
	ObjectType		: E_BACNETOBJECTTYPE;
	ObjectInstance	: UDINT;
END_VAR
VAR
END_VAR
F_BACnet_GetObjId := F_BACnet_GetObjInstance(ObjectInstance) + SHL(INT_TO_UDINT(ObjectType), 22);
END_FUNCTION

(* POU F_BACnet_GetStatusFlagsData, ST *)
FUNCTION F_BACnet_GetStatusFlagsData : WORD
VAR_INPUT
	Flags : ST_BACnet_StatusFlags;
END_VAR
F_BACnet_GetStatusFlagsData	:= 16#0004;
IF Flags.in_alarm THEN
	F_BACnet_GetStatusFlagsData := DWORD_TO_WORD(_F_BACnet_SetBitFieldBit(ptrData:=ADR(F_BACnet_GetStatusFlagsData), Bit:=BACnetStatusFlags_in_alarm));
END_IF
IF Flags.fault THEN
	F_BACnet_GetStatusFlagsData := DWORD_TO_WORD(_F_BACnet_SetBitFieldBit(ptrData:=ADR(F_BACnet_GetStatusFlagsData), Bit:=BACnetStatusFlags_fault));
END_IF
IF Flags.overridden THEN
	F_BACnet_GetStatusFlagsData := DWORD_TO_WORD(_F_BACnet_SetBitFieldBit(ptrData:=ADR(F_BACnet_GetStatusFlagsData), Bit:=BACnetStatusFlags_overridden));
END_IF
IF Flags.out_of_service THEN
	F_BACnet_GetStatusFlagsData := DWORD_TO_WORD(_F_BACnet_SetBitFieldBit(ptrData:=ADR(F_BACnet_GetStatusFlagsData), Bit:=BACnetStatusFlags_out_of_service));
END_IF
END_FUNCTION

(* POU F_BACnet_IsFinite, ST *)
FUNCTION F_BACnet_IsFinite : BOOL
VAR_INPUT
	fValue		: REAL;
END_VAR
VAR
	fArg		: T_Arg;
END_VAR
fArg.cbLen := SIZEOF(fValue);
fArg.eType := ARGTYPE_REAL;
fArg.pData := ADR(fValue);
F_BACnet_IsFinite := IsFinite(fArg);
END_FUNCTION

(* POU F_BACnet_LimitEnableFlags, ST *)
FUNCTION F_BACnet_LimitEnableFlags : ST_BACnet_LimitEnable
VAR_INPUT
	data	: WORD;
END_VAR
VAR
END_VAR
F_BACnet_LimitEnableFlags.highLimitEnable := _F_BACnet_IsBitFieldBitSet( data:=data, Bit:=BACnetLimitEnableBits_highLimit);
F_BACnet_LimitEnableFlags.lowLimitEnable := _F_BACnet_IsBitFieldBitSet( data:=data, Bit:=BACnetLimitEnableBits_lowLimit);
END_FUNCTION

(* POU F_BACnet_MultiStatePV, ST *)
FUNCTION F_BACnet_MultiStatePV : UDINT
VAR_INPUT
	bEnable	: BOOL; (* TRUE = commit to stack, FALSE = do-nothing *)
	bNull	: BOOL; (* TRUE = clear priority, FALSE = write number from state input *)
	nState	: UDINT; (* multi-state [1..max-number-of-states] *)
END_VAR
IF (bEnable) THEN
	IF (bNull) THEN
		F_BACnet_MultiStatePV := 16#0;
	ELSE
		F_BACnet_MultiStatePV := nState;
	END_IF
ELSE
	F_BACnet_MultiStatePV := 16#FFFFFFFF;
END_IF
END_FUNCTION

(* POU F_BACnet_RealEQ, ST *)
FUNCTION F_BACnet_RealEQ : BOOL
VAR_INPUT
	fIn1	: REAL;
	fIn2	: REAL;
END_VAR
VAR
END_VAR
IF (F_BACnet_IsFinite(fIn1) <> F_BACnet_IsFinite(fIn2)) THEN
	F_BACnet_RealEQ := FALSE;
	RETURN;
END_IF
IF F_BACnet_IsFinite(fIn1) THEN
	IF (fIn1 <> fIn2) THEN
		F_BACnet_RealEQ := FALSE;
		RETURN;
	END_IF
END_IF
F_BACnet_RealEQ := TRUE;
END_FUNCTION

(* POU F_BACnet_RealGE, ST *)
FUNCTION F_BACnet_RealGE : BOOL
VAR_INPUT
	fIn1	: REAL;
	fIn2	: REAL;
END_VAR
VAR
END_VAR
IF NOT (F_BACnet_IsFinite(fIn1) OR F_BACnet_IsFinite(fIn2)) THEN
	F_BACnet_RealGE := FALSE;
	RETURN;
END_IF
F_BACnet_RealGE := (fIn1 >= fIn2);
END_FUNCTION

(* POU F_BACnet_RealGT, ST *)
FUNCTION F_BACnet_RealGT : BOOL
VAR_INPUT
	fIn1	: REAL;
	fIn2	: REAL;
END_VAR
VAR
END_VAR
IF NOT (F_BACnet_IsFinite(fIn1) OR F_BACnet_IsFinite(fIn2)) THEN
	F_BACnet_RealGT := FALSE;
	RETURN;
END_IF
F_BACnet_RealGT := (fIn1 > fIn2);
END_FUNCTION

(* POU F_BACnet_RealLE, ST *)
FUNCTION F_BACnet_RealLE : BOOL
VAR_INPUT
	fIn1	: REAL;
	fIn2	: REAL;
END_VAR
VAR
END_VAR
IF NOT (F_BACnet_IsFinite(fIn1) OR F_BACnet_IsFinite(fIn2)) THEN
	F_BACnet_RealLE := FALSE;
	RETURN;
END_IF
F_BACnet_RealLE := (fIn1 <= fIn2);
END_FUNCTION

(* POU F_BACnet_RealLT, ST *)
FUNCTION F_BACnet_RealLT : BOOL
VAR_INPUT
	fIn1	: REAL;
	fIn2	: REAL;
END_VAR
VAR
END_VAR
IF NOT (F_BACnet_IsFinite(fIn1) OR F_BACnet_IsFinite(fIn2)) THEN
	F_BACnet_RealLT := FALSE;
	RETURN;
END_IF
F_BACnet_RealLT := (fIn1 < fIn2);
END_FUNCTION

(* POU F_BACnet_RealNothing, ST *)
FUNCTION F_BACnet_RealNothing : DWORD
F_BACnet_RealNothing:=16#7FFFFFFF;
END_FUNCTION

(* POU F_BACnet_RealPV, ST *)
FUNCTION F_BACnet_RealPV : DWORD
VAR_INPUT
	bEnable	: BOOL; (* TRUE = commit to stack, FALSE = do-nothing *)
	bNull	: BOOL; (* TRUE = clear priority, FALSE = write value from input *)
	rValue	: REAL;
END_VAR
VAR
	pDword : POINTER TO DWORD;
END_VAR
IF (bEnable) THEN
	IF (bNull) THEN
		F_BACnet_RealPV := F_BACnet_RealNull();
	ELSE
		pDword := ADR(rValue);
		F_BACnet_RealPV := pDword^;
	END_IF
ELSE
	F_BACnet_RealPV := F_BACnet_RealNothing();
END_IF
END_FUNCTION

(* POU F_BACnet_RealToStr, ST *)
FUNCTION F_BACnet_RealToStr : STRING
VAR_INPUT
	pValue	: POINTER TO REAL;
END_VAR
VAR
	fArg	: T_Arg;
	pDWORD	: POINTER TO DWORD;
END_VAR
fArg.cbLen := 4;
fArg.eType := ARGTYPE_REAL;
fArg.pData := pValue;
pDWORD := pValue;
IF IsFinite(fArg) THEN
	F_BACnet_RealToStr := REAL_TO_STRING(pValue^);
ELSE
	IF (pDWORD^ = 16#7FFF0000) THEN
		F_BACnet_RealToStr := '#NULL';
	ELSIF (pDWORD^ AND 16#80000000) = 16#80000000 THEN
		F_BACnet_RealToStr := '-#QNAN';
	ELSE
		F_BACnet_RealToStr := '#QNAN';
	END_IF
END_IF
END_FUNCTION

(* POU F_BACnet_StatusFlags, ST *)
FUNCTION F_BACnet_StatusFlags : ST_BACnet_StatusFlags
VAR_INPUT
	data	: WORD;
END_VAR
VAR
END_VAR
F_BACnet_StatusFlags.in_alarm:= _F_BACnet_IsBitFieldBitSet( data:=data, Bit:=BACnetStatusFlags_in_alarm);
F_BACnet_StatusFlags.fault:= _F_BACnet_IsBitFieldBitSet( data:=data, Bit:=BACnetStatusFlags_fault);
F_BACnet_StatusFlags.overridden:= _F_BACnet_IsBitFieldBitSet( data:=data, Bit:=BACnetStatusFlags_overridden);
F_BACnet_StatusFlags.out_of_service:= _F_BACnet_IsBitFieldBitSet( data:=data, Bit:=BACnetStatusFlags_out_of_service);
END_FUNCTION

(* POU F_BACnet_TimeHasPlaceholder, ST *)
FUNCTION F_BACnet_TimeHasPlaceholder : BOOL
VAR_INPUT
	stTime		: ST_BACnet_Time;
END_VAR
F_BACnet_TimeHasPlaceholder := (stTime.nHour = 16#FF) OR (stTime.nHundredths = 16#FF) OR (stTime.nMinute = 16#FF) OR (stTime.nSecond = 16#FF);
END_FUNCTION

(* POU F_BACnet_TimeMerge, ST *)
FUNCTION F_BACnet_TimeMerge : ST_BACnet_Time (* This function replaces placeholder in time1 with time2 and returning the result (if no placeholder is given, time1 will be prefered) *)
VAR_INPUT
	stTime1		: ST_BACnet_Time;
	stTime2		: ST_BACnet_Time;
END_VAR
VAR
END_VAR
IF stTime1.nHour = 16#FF THEN
	F_BACnet_TimeMerge.nHour := F_BACnet_CheckHour(stTime2.nHour);
ELSE
	F_BACnet_TimeMerge.nHour := F_BACnet_CheckHour(stTime1.nHour);
END_IF
IF stTime1.nHundredths = 16#FF THEN
	F_BACnet_TimeMerge.nHundredths := F_BACnet_CheckHundredths(stTime2.nHundredths);
ELSE
	F_BACnet_TimeMerge.nHundredths := F_BACnet_CheckHundredths(stTime1.nHundredths);
END_IF
IF stTime1.nMinute = 16#FF THEN
	F_BACnet_TimeMerge.nMinute := F_BACnet_CheckMinute(stTime2.nMinute);
ELSE
	F_BACnet_TimeMerge.nMinute := F_BACnet_CheckMinute(stTime1.nMinute);
END_IF
IF stTime1.nSecond = 16#FF THEN
	F_BACnet_TimeMerge.nSecond := F_BACnet_CheckSecond(stTime2.nSecond);
ELSE
	F_BACnet_TimeMerge.nSecond := F_BACnet_CheckSecond(stTime1.nSecond);
END_IF
END_FUNCTION

(* POU F_BACnet_TimeStruct_TO_DateTime, ST *)
FUNCTION F_BACnet_TimeStruct_TO_DateTime : ST_BACnet_DateTime
VAR_INPUT
	IN	: TIMESTRUCT;
END_VAR
F_BACnet_TimeStruct_TO_DateTime.stDate.nDay			:= WORD_TO_BYTE(IN.wDay);
IF IN.wDayOfWeek = 0 THEN
	F_BACnet_TimeStruct_TO_DateTime.stDate.nDayOfWeek := 7;
ELSE
	F_BACnet_TimeStruct_TO_DateTime.stDate.nDayOfWeek := WORD_TO_BYTE(IN.wDayOfWeek);
END_IF
F_BACnet_TimeStruct_TO_DateTime.stDate.nMonth		:= WORD_TO_BYTE(IN.wMonth);
F_BACnet_TimeStruct_TO_DateTime.stDate.nYear		:= WORD_TO_BYTE(IN.wYear - 1900);
F_BACnet_TimeStruct_TO_DateTime.stTime.nHour		:= WORD_TO_BYTE(IN.wHour);
F_BACnet_TimeStruct_TO_DateTime.stTime.nMinute		:= WORD_TO_BYTE(IN.wMinute);
F_BACnet_TimeStruct_TO_DateTime.stTime.nSecond		:= WORD_TO_BYTE(IN.wSecond);
F_BACnet_TimeStruct_TO_DateTime.stTime.nHundredths	:= WORD_TO_BYTE(IN.wMilliseconds / 10);
END_FUNCTION

(* POU F_BACnet_TimeUnspecified, ST *)
FUNCTION F_BACnet_TimeUnspecified : BOOL
VAR_INPUT
	stTime		: ST_BACnet_Time;
END_VAR
F_BACnet_TimeUnspecified := (stTime.nHour = 16#FF) AND (stTime.nHundredths = 16#FF) AND (stTime.nMinute = 16#FF) AND (stTime.nSecond = 16#FF);
END_FUNCTION

(* POU F_BinPV_AND, ST *)
FUNCTION F_BinPV_AND : E_BACNETBINARYPV
VAR_INPUT
	eBinPV1:	E_BACNETBINARYPV;
	eBinPV2:	E_BACNETBINARYPV;
END_VAR
VAR
END_VAR
IF (eBinPV1 = eBinPV2) THEN
	F_BinPV_AND := eBinPV1;
ELSE
	F_BinPV_AND := BACnetBinaryPV_Nothing;
END_IF
END_FUNCTION

(* POU F_BinPV_NOT, ST *)
FUNCTION F_BinPV_NOT : E_BACNETBINARYPV
VAR_INPUT
	eBinPV:	E_BACNETBINARYPV;
END_VAR
VAR
END_VAR
IF (eBinPV = BACnetBinaryPV_active) THEN
	F_BinPV_NOT := BACnetBinaryPV_inactive;
ELSIF (eBinPV = BACnetBinaryPV_inactive) THEN
	F_BinPV_NOT := BACnetBinaryPV_active;
ELSE
	F_BinPV_NOT := eBinPV;
END_IF
END_FUNCTION

(* POU F_BinPV_OR, ST *)
FUNCTION F_BinPV_OR : E_BACNETBINARYPV
VAR_INPUT
	eBinPV1:	E_BACNETBINARYPV;
	eBinPV2:	E_BACNETBINARYPV;
END_VAR
VAR
END_VAR
IF (eBinPV1 = BACnetBinaryPV_active) OR (eBinPV2 = BACnetBinaryPV_active) THEN
	F_BinPV_OR := BACnetBinaryPV_active;
ELSIF (eBinPV1 = BACnetBinaryPV_inactive) OR (eBinPV2 = BACnetBinaryPV_inactive) THEN
	F_BinPV_OR := BACnetBinaryPV_inactive;
ELSIF (eBinPV1 = BACnetBinaryPV_NULL) OR (eBinPV2 = BACnetBinaryPV_NULL) THEN
	F_BinPV_OR := BACnetBinaryPV_NULL;
ELSE
	F_BinPV_OR := BACnetBinaryPV_Nothing;
END_IF
END_FUNCTION

(* POU F_BinPV_To_Bool, ST *)
FUNCTION F_BinPV_To_Bool : BOOL
VAR_INPUT
	eBinPV		: E_BACNETBINARYPV;
END_VAR
VAR
END_VAR
F_BinPV_To_Bool := (eBinPV = BACnetBinaryPV_active);
END_FUNCTION

(* POU F_BinPV_XOR, ST *)
FUNCTION F_BinPV_XOR : E_BACNETBINARYPV
VAR_INPUT
	eBinPV1:	E_BACNETBINARYPV;
	eBinPV2:	E_BACNETBINARYPV;
END_VAR
VAR
END_VAR
IF (eBinPV1 = BACnetBinaryPV_active) XOR (eBinPV2 = BACnetBinaryPV_active) THEN
	F_BinPV_XOR := BACnetBinaryPV_active;
ELSIF (eBinPV1 = BACnetBinaryPV_inactive) XOR (eBinPV2 = BACnetBinaryPV_inactive) THEN
	F_BinPV_XOR := BACnetBinaryPV_inactive;
ELSIF (eBinPV1 = BACnetBinaryPV_NULL) XOR (eBinPV2 = BACnetBinaryPV_NULL) THEN
	F_BinPV_XOR := BACnetBinaryPV_NULL;
ELSE
	F_BinPV_XOR := BACnetBinaryPV_Nothing;
END_IF
END_FUNCTION

(* POU F_Bool_To_BinPV, ST *)
FUNCTION F_Bool_To_BinPV : E_BACNETBINARYPV
VAR_INPUT
	bEnable	: BOOL;
	bNull	: BOOL;
	bBool	: BOOL;
END_VAR
VAR
END_VAR
IF (NOT bEnable) THEN
	F_Bool_To_BinPV := BACnetBinaryPV_Nothing;
ELSIF bNull THEN
	F_Bool_To_BinPV := BACnetBinaryPV_NULL;
ELSIF bBOOL THEN
	F_Bool_To_BinPV := BACnetBinaryPV_active;
ELSE
	F_Bool_To_BinPV := BACnetBinaryPV_inactive;
END_IF
END_FUNCTION

(* POU F_GetVersionTcBACnet, ST *)
FUNCTION F_GetVersionTcBACnet : UINT		(* Gets the library version info *)
VAR_INPUT
	nVersionElement		: INT;
END_VAR


(* Possible nVersionElement number:
	1	:	major number
	2	:	minor number
	3	: 	revision number
*)

(* Version history:
Date		|	Version/Author			|	Created with				|	Remark
-----------------------------------------------------------------------------------------------------------------------------------
13/03/12	|	1.0.0	/ MAr			|	V2.11.0 (Build 2218)		|	* Renamed BACnet-datatype ENUM entries
20/03/12	|	1.1.0	/ MAr			|	V2.11.0 (Build 2219)		|	* Added new function blocks with ADS property write support (for WOC on local objects present_value)
			|							|								|	* Added optional input to FB_BACnet_Device to setup the valid ADS port (default 1000)
20/03/12	|	1.1.1	/ MAr			|	V2.11.0 (Build 2219)		|	* Removed obsolete flags in FB_BACnet_Program function block
27/03/12	|	1.1.2	/ MAr			|	V2.11.0 (Build 2219)		|	* FB_BACnet_ReadProp returns real processed data len (nProcessedLen)
			|							|								|	* new helper function "F_BACnet_GetObjId" added
28/03/12	|	1.1.3	/ MAr			|	V2.11.0 (Build 2219)		|	* fixed error reset in "FB_BACnet_Device"
			|							|								|	* filter object instance number in "F_BACnet_GetObjId" to prevent overflow
			|							|								|	* added ending element of BACnetObjectType-Enumeration
			|							|								|	* renamed "bErrorId" to "nErrorId" in "FB_BACnet_NotificationSinkDelEntry"
10/04/12	|	1.1.4	/ MAr			|	V2.11.0 (Build 2220)		|	* FB_BACnet_ReadProp extended with automatic handling for range properties (READ_RANGE)
21/05/12	|	1.2.0	/ MAr			|	V2.11.0 (Build 2222)		|	* Changed ENUM names to capital letter (upper case)
			|							|								|	* Renamed LOOP object process data "_SystemStatus" to "_PresentValueI"
			|							|								|	* Append update logic for remote device into remote object FBs (no need to call remote device FB explicit)
29/05/12	|	1.2.1	/ MAr			|	V2.11.0 (Build 2223)		|	* Append local object for Accumulator access (and also _EX version)
20/07/12	|	1.2.2	/ MAr			|	V2.11.0 (Build 2224)		|	* New kind of BACnet FBs "_RAW" for read/write raw values in PLC program instead of direct hardware link
			|							|								|	* Added "AckedTransitions" flags to "_EX" function blocks
			|							|								|	* Added automatic client reset to FB_BACnet_RemoteDevice (timeouts will counted, but didn't interrupt client functionality if auto-reset is active)
			|							|								|	* New time out counter as output status to FB_BACnet_RemoteDevice added
23/07/12	|	1.2.3	/ MAr			|	V2.11.0 (Build 2226)		|	* Added service fail counter to FB_BACnet_RemoteDevice
20/12/12	|	1.3.0	/ MAr	(Beta)	|	V2.11.0 (Build 2232)		|	* Added ADS-Connection blocks (easy to connect objects over ADS)
			|							|								|	* Added local object function blocks with revision 9 features (BETA versions!)
			|							|								|	* Major-change in exisiting object: FB_BACnet_Loop object dosn't write "OutOfService" anymore
			|							|								|	* New raw version of the ACC object type
			|							|								|	* Added flag helper functions
20/12/12	|	1.3.1	/ MAr	(Beta)	|	V2.11.0 (Build 2232)		|	* Optimized error handling for remote device
			|							|								|	* auto detect legacy mode in remote device and fill AdsConn infos from remote device inputs
08/07/13	|	1.3.2	/ MAr	(Beta)	|	V2.11.0 (Build 2234)		|	* added missing _RAW types to R9
21/08/13	|	1.3.3	/ MAr			|	V2.11.0 (Build 2234)		|	* added new function block for time synchronization over BACnet (local time --> BACnet server --> BACnet broadcast)
06/09/13	|	2.0.0	/ MAr			|	V2.11.0 (Build 2234)		|	* removed legacy function blocks and replaced with R9 versions
			|							|								|	* added function blocks for property access
			|							|								|	* error codes are complete global now
			|							|								|	* optimized process data (removed object ID for basic FBs, sorted process data with focus on alignment)
10/09/13	|	2.0.1	/ MAr			|	V2.11.0 (Build 2237)		|	* new function block for EE object add
02/10/13	|	2.0.2	/ MAr			|	V2.11.0 (Build 2237)		|	* Mapped LocalTime and -Date into Device object
			|							|								|	* Added some helper and signal functions
			|							|								|	* PID auto tuning added into LOOP_EX version
			|							|								|	* Added LOOP objects using internal stack LOOP controller (performance optimized)
			|							|								|	* Removed obsolete function blocks
05/11/13	|	2.0.3	/ MAr			|	V2.11.0 (Build 2237)		|	* Added Multi-State objects as RAW-type
			|							|								|	* Renamed BACnetInfo structure member
			|							|								|	* Added feedback and error flag to RAW function blocks
			|							|								|	* First cycle flag moved on first position in function block logic
			|							|								|	* added WOC-disable service and PLC-startup flag into device object
			|							|								|	* clear data buffer in ReadProp function block (because client data optimized and size of read data maybe lower than buffer size)
19/03/14	|	2.0.4	/ MAr			|	V2.11.0 (Build 2240)		|	* removed obsolete check
10/04/14	|	2.1.0	/ MAr			|	V2.11.0 (Build 2241)		|	* PLC ready flag delayed by device status
23/04/14	|	2.2.0	/ MAr			|	V2.11.0 (Build 2241)		|	* Removed "POLL" version of remote FBs (poll mode can be configured by function block comments)
			|							|								|	* Changed default present_value of object function blocks to "do-nothing"
			|							|								|	  (NULL is furthermore writeable by F_BACnet_RealNull or special Binary-PV [2] or multi-state [0] values)
			|							|								|	* Added new function blocks for PV values (F_BACnet_AnalogPV and F_BACnet_MultiStatePV)
			|							|								|	* Added "a-life" bit to remote device function block
20/05/14	|	2.2.1	/ MAr			|	V2.11.0 (Build 2241)		|	* Fixed "ReadMessageTexts"
			|							|								|	* Default value for command object changed to 0x0 instead 0xffffffff
02/06/14	|	2.2.2	/ MAr			|	V2.11.0 (Build 2241)		|	* Added Notification-Sink read and remove functions (Rev. 12 and above only)
			|							|								|	* Added Notification-Sink function block
			|							|								|	* optimized encoding function (when source and target are diffent memory areas with same byte size)
11/06/14	|	2.2.3	/ MAr			|	V2.11.0 (Build 2241)		|	* Added "bReload" input into local and remote device object
			|							|								|	* automatic LOOP mode detection (ideal mode vs. standard mode) according to the property unit of integral_ and derivative_constant
			|							|								|		- ideal mode means: clear parallel junktion of P, I and D (parameter Kp, Ki and Kd are gain [1] constants for each element)
			|							|								|		- standard mode means: serial junktion of P and I parallel to P and D (parameter Kp is the gain constant [1], Ti and Td are time based [s])
14/11/14	|	2.2.4	/ MAr			|	V2.11.0 (Build 2245)		|	* Added stValidFields into Notification-Event structure
			|							|								|	* Optimized STRING conversion for Object-ID and Date/Time
			|							|								|	* Optimized result type for F_BACnet_GetObjId
20/11/14	|	2.2.5	/ MAr			|	V2.11.0 (Build 2245)		|	* Optimized data handling for Log_Buffer property function block
05/12/14	|	2.2.6	/ MAr			|	V2.11.0 (Build 2245)		|	* Optimized process data default value for remote program object
16/01/15	|	2.2.7	/ MAr			|	V2.11.0 (Build 2245)		|	* New function for "Nothing" process data coding for analog* objects
19/01/15	|	2.3.0	/ MAr			|	V2.11.0	(Build 2245)		|	* Changed default FB to read-only (except local LOOP and PROG)
			|							|								|	* Append new "_WR" function block types to enable write access for commandable basic function blocks (remote and local)
23/01/15	|	2.3.1	/ MAr			|	V2.11.0	(Build 2245)		|	* Optimize value compare in ADS-type of analog* objects
10/02/15	|	2.4.0	/ MAr			|	V2.11.0	(Build 2245)		|	* Remove local _WR-Object types
23/10/15	|	2.4.1	/ MAr			|	V2.11.0 (Build 2248)		|	* Added exception- and weekly-schedule property with REAL value capability
04/11/15	|	2.4.2	/ MAr			|	V2.11.0 (Build 2248)		|	* Fixed data type handling in new REAL type properties
06/11/15	|	2.4.3	/ MAr			|	V2.11.0 (Build 2248)		|	* Fallback for PID mode, if property I or D is deactivated
12/02/16	|	2.4.4	/ MAr			|	V2.11.0 (Build 2269)		|	* removed restricted status check in remote device object
14/04/16	|	2.4.5	/ MAr			|	V2.11.0 (Build 2254)		|	* changed input parameter type of FB_BACnet_AvgValue (UINT --> INT)
18/04/16	|	2.5.0	/ MAr			|	V2.11.0 (Build 2254)		|	* Added TrendLogMultiple and EventLog Objects (standard, EX and remote)
*)
CASE nVersionElement OF
	1:	F_GetVersionTcBACnet := 2;
	2:	F_GetVersionTcBACnet := 5;
	3:	F_GetVersionTcBACnet := 0;
	ELSE
		F_GetVersionTcBACnet := 16#FFFF;
END_CASE
END_FUNCTION

(* POU FB_BACnet_AccLimit, ST *)
FUNCTION_BLOCK FB_BACnet_AccLimit
VAR_INPUT
	X : REAL; (* input value [1] *)
	Amax : REAL; (* maximum acceleration of X [1/s]; 0 = limit disabled *)
	Tcycle : REAL; (* cycle time [s] of task; 0 = use internal measuring *)
END_VAR
VAR_OUTPUT
	Y : REAL; (* limited X value [1] *)
	A : REAL; (* input acceleration [1/s] *)
END_VAR
VAR
	_sysTime	: GETCPUCOUNTER;
	_Time		: T_LARGE_INTEGER;
	_TimeOld	: T_LARGE_INTEGER;
	_cycleTime	: REAL;
	_bFirstScan	: BOOL:=TRUE;
	_foldY		: REAL;
END_VAR
(* determine cycle time *)
IF Tcycle = 0.0 THEN
	_TimeOld := _Time;
	_sysTime(cpuCntLoDW=> _Time.dwLowPart, cpuCntHiDW=> _Time.dwHighPart);
	_cycleTime := _F_BACnet_SysTimeDiff(In1:=_Time, In2:=_TimeOld);
ELSE
	_cycleTime := Tcycle;
END_IF

IF (NOT _bFirstScan) THEN
	(* exit on wrong cycle time *)
	IF _cycleTime <= 0.0 THEN
		RETURN;
	END_IF
	(* calculate current acceleration *)
	A := (X - _foldY) / _cycleTime;
	IF (Amax <> 0.0) THEN
		Amax := ABS(Amax);
		IF (ABS(A) > Amax) THEN
			IF (A >= 0.0) THEN
				Y := _foldY + (Amax * _cycleTime);
			ELSE
				Y := _foldY - (Amax * _cycleTime);
			END_IF
		ELSE
			Y := X;
		END_IF
	ELSE
		Y := X;
	END_IF
ELSE
	Y := X;
END_IF

_foldY := Y;
_bFirstScan:=FALSE;
END_FUNCTION_BLOCK

(* POU FB_BACnet_Accumulator, ST *)
FUNCTION_BLOCK FB_BACnet_Accumulator
VAR_INPUT
	nValueSet			: UDINT; (* number for present_value *)
END_VAR
VAR_IN_OUT
	Device				: FB_BACnet_Device;
END_VAR
VAR_OUTPUT
	bReady				: BOOL;
	nPresentValue		: UDINT;
	bOverridden			: BOOL;
	bOutOfService		: BOOL;
	bFault				: BOOL;
	bInAlarm			: BOOL;
	bError				: BOOL;
	nErrorId			: UINT;
END_VAR
VAR
	_PresentValueIn AT%I*:UDINT;	(* ~(BACnet_PresentValue	:		: )
										(BACnet_MaxPresValue	:		: writeprotect,nolink)
										(BACnet_ObjectType		: ACC	: )	*)
	_ValueSet AT%Q*:UDINT;			(* ~(BACnet_ValueSet		:		: ) *)
	_StatusFlags AT%I*:WORD;		(* ~(BACnet_StatusFlags		:		: )	*)
	_StatusFlagsBits : ST_BACnet_StatusFlags;

	_nUpdateCount : UDINT := 0;
END_VAR
(* update device *)
IF Device._nUpdateCount = _nUpdateCount THEN
	Device();
END_IF
(* remind current number of update counter *)
_nUpdateCount := Device._nUpdateCount;

IF _StatusFlags < 4 THEN
	(* mapping seems to be wrong (bit string for status flags must be 4 in minimum) *)
	nErrorId := BACnet_ERR_WRONG_MAPPING;

ELSIF Device.bOperational THEN
	(* clear error flag *)
	nErrorId := BACnet_ERR_NO_ERROR;
	bReady := TRUE;
	(* copy present value *)
	nPresentValue 		:= _PresentValueIn;
	_ValueSet			:= nValueSet;

	(* build bit states *)
	_StatusFlagsBits	:= F_BACnet_StatusFlags(_StatusFlags);

	(* copy states to output *)
	bOverridden := _StatusFlagsBits.overridden;
	bOutOfService := _StatusFlagsBits.out_of_service;
	bFault := _StatusFlagsBits.fault;
	bInAlarm := _StatusFlagsBits.in_alarm;
ELSE
	bReady := FALSE;
	(* and set error ID *)
	nErrorId := BACnet_ERR_OPERATIONAL;
END_IF

(* set error flag *)
bError := (nErrorId <> BACnet_ERR_NO_ERROR);
END_FUNCTION_BLOCK

(* POU FB_BACnet_Device, ST *)
FUNCTION_BLOCK FB_BACnet_Device
VAR_INPUT
	bReset				: BOOL; (* reset errors *)
	bSupportBackup		: BOOL; (* support backup of PLC persistent data when BACnet backup service is used *)
	bWritePersis		: BOOL; (* Manual trigger for PLC and BACnet persistent data storage *)
	bDisableWOC			: BOOL; (* Deactivate write-on-change mechanism *)
	bReload				: BOOL; (* Reload ADS connection and increase reload counter (trigger autoget) *)
	nAmsPort			: T_AmsPort := 1000; (* default port when port can not be determined automatically *)
END_VAR
VAR_OUTPUT
	nRevision			: DINT := -1; (* protocol revision no. *)
	stAdsConn			: ST_BACnet_AdsConnection;
	eSystemStatus		: E_BACNETDEVICESTATUS;
	bBackupActive		: BOOL;
	bWritePersisActive	: BOOL;
	bOperational		: BOOL;
	bWOCDisabled		: BOOL;
	bFirstCycle			: BOOL;
	dtLocalTime			: ST_BACnet_DateTime;
	bError				: BOOL;
	nErrorId			: UINT;
END_VAR
VAR
	_ObjectId			AT%I*: DWORD;	(* ~(BACnet_ObjectIdentifier:		: LINK) *)
	_LocalDate			AT%I*: DWORD;	(* ~(BACnet_LocalDate		:		: LINK) *)
	_LocalTime			AT%I*: DWORD;	(* ~(BACnet_LocalTime		:		: LINK) *)
	_SystemStatus		AT%I*: WORD;	(* ~(BACnet_SystemStatus	:		: )
								   			(BACnet_ObjectType		: DEV	: )	*)
	_ServerStatus		AT%I*: WORD;	(* ~(BACnet_ServerStatus	:		: )	*)
	_ServerControl		AT%Q*: WORD;	(* ~(BACnet_ServerControl	:		: )	*)
	_fbWritePersistent	: FB_WritePersistentData;
	_rtrigBackup		: R_TRIG;
	_rtrigReset			: R_TRIG;

	_bHasStarted		: BOOL := TRUE;
	_nPlcPort			: T_AmsPort;

	_nUpdateCount	 	: UDINT := 0;
	_nUpdateCountAdp 	: UDINT := 0;
	_BACnetAdapter		: POINTER TO FB_BACnet_Adapter;
	_AdsConn			: _FB_BACnet_AdsConn;
	_WritePersistentProp: FB_BACnet_WriteProp;
	_ReadPersistentProp	: FB_BACnet_ReadProp;
	_iPersis			: INT;
	_nPersistentState	: DWORD;
	_ePersistentState	: E_BACNETPERSISTENTDATASTATE;
	_tonPersisTimeout	: TON;
	_tonPersisPoll		: TON;
	_bPersisWritten		: BOOL;
	_ReadRevisionProp	: FB_BACnet_ReadProp;
	_iRevision			: INT;
	_pLocalDate			: POINTER TO ST_BACnet_Date;
	_pLocalTime			: POINTER TO ST_BACnet_Time;
END_VAR
(* check pointer to bacnet adapter instance *)
IF pBACnet_Adapter > 0 THEN
	_BACnetAdapter := pBACnet_Adapter;
ELSE
	_BACnetAdapter := ADR(fbBACnet_Adapter);
END_IF

(* update adapter *)
IF _BACnetAdapter^._nUpdateCount = _nUpdateCountAdp THEN
	_BACnetAdapter^();
END_IF
(* remind current number of update counter *)
_nUpdateCountAdp := _BACnetAdapter^._nUpdateCount;

(* convert SystemStatus to enumeration *)
eSystemStatus := _SystemStatus;

(* reset trigger *)
_rtrigReset(CLK:= bReset, Q=> );
(* reset error ID and flag *)
IF (nErrorId < 20) OR (nErrorId >= 30) OR _rtrigReset.Q THEN
	nErrorId := BACnet_ERR_NO_ERROR;
END_IF

(* check if NetID is plausible *)
IF _BACnetAdapter^.sAmsNetId = '' THEN
	(* NetId not OK, return with error *)
	nErrorId := BACnet_ERR_NO_VALID_NET_ID;
END_IF

IF ((bSupportBackup) OR (_fbWritePersistent.START AND (_iPersis = 0))) THEN
	(* PLC can be backup't *)
	_ServerControl.0 := TRUE;
ELSE
	(* don't support PLC backup *)
	_ServerControl.0 := FALSE;
	_ServerControl.1 := FALSE;
END_IF

(* trigger backup flag *)
_rtrigBackup(CLK:= (eSystemStatus = BACnetDeviceStatus_BackupInProgress) AND (_iPersis = 0), Q=> );
IF (_iPersis = 0) THEN
	(* only backup if persistent state machine is idle *)
	IF _rtrigBackup.Q AND _ServerControl.0 THEN
		(* trigger backup function *)
		_fbWritePersistent.START := TRUE;
	ELSIF _fbWritePersistent.START AND (NOT _fbWritePersistent.BUSY) THEN
		IF _fbWritePersistent.ERR THEN
			(* backup aborted *)
			nErrorId := BACnet_ERR_PERSISTENT_PLC_WRITE;
		ELSE
			(* backup was successful *)
			_ServerControl.1 := TRUE;
		END_IF
	ELSIF (eSystemStatus <> BACnetDeviceStatus_BackupInProgress) THEN
		(* backup process finished *)
		_ServerControl.1 := FALSE;
	END_IF
END_IF

(* calculate PLC runtime port *)
_nPlcPort := ((SystemInfo.runTimeNo - 1) * 10) + SystemInfo.runTimeNo + 800;

(* call persistent backup *)
_fbWritePersistent(
	NETID	:= '',
	PORT	:= _nPlcPort,
	START	:= ,
	TMOUT	:= BACnet_PlcPersisTimeOut,
	MODE	:= SPDM_VAR_BOOST,
	BUSY	=> ,
	ERR		=> ,
	ERRID	=>
);

(* call ADS connection *)
IF (_ObjectId <> 16#00000000) THEN
	_AdsConn(
		bAutoReload		:= bOperational,
		bReload			:= 	(bReset AND (NOT _AdsConn.bReady))
						OR	bReload,
		bDevOperational	:= bOperational,
		sAmsNetId		:= _BACnetAdapter^.sAmsNetId,
		tDevObjId		:= _ObjectId,
		bIsClient		:= FALSE,
		bReady			=> ,
		bBusy			=> ,
		bDone			=> ,
		bError			=> ,
		nErrorId		=> ,
		stBACnetAds		=> );
END_IF

(* error when ADS connection failed *)
IF _AdsConn.bError THEN
	IF (_AdsConn.nErrorId = BACnet_ERR_ADS_LegacyStack) THEN
		nRevision := 6;
		stAdsConn.bServer := TRUE;
		stAdsConn.bClient := FALSE;
		IF		(NOT stAdsConn.bValid)
			OR	(stAdsConn.nDeviceId <> F_BACnet_GetObjInstance(_ObjectId))
			OR	(stAdsConn.nAmsPort <> nAmsPort)
			OR	(stAdsConn.sAmsNetId <> _BACnetAdapter^.sAmsNetId)
		THEN
			stAdsConn.nReload := stAdsConn.nReload + 1;
		END_IF
		stAdsConn.nDeviceId	:= F_BACnet_GetObjInstance(_ObjectId);
		stAdsConn.sAmsNetId	:= _BACnetAdapter^.sAmsNetId;
		stAdsConn.nAmsPort	:= nAmsPort;
		stAdsConn.bValid	:= TRUE;
	ELSE
		IF (nErrorId = 0) THEN
			nErrorId	:= _AdsConn.nErrorId;
		END_IF
		nRevision := -1;
		stAdsConn	:= _AdsConn.stBACnetAds;
	END_IF
ELSIF _AdsConn.bDone THEN
	stAdsConn := _AdsConn.stBACnetAds;
ELSIF (NOT _AdsConn.bReady) THEN
	nRevision := -1;
END_IF

(* read revision no. *)
_ReadRevisionProp(
	BACnetDevicePort:= stAdsConn.nAmsPort,
	bExecute		:= ,
	sNetId			:= stAdsConn.sAmsNetId,
	ObjectType		:= BACnetObjectType_Device,
	PropertyID		:= BACnetPropertyIdentifier_ProtocolRevision,
	DataType		:= BACnetDataType_UnsignedInteger,
	ObjectInstance	:= stAdsConn.nDeviceId,
	ptrValue		:= ADR(nRevision),
	nLenValue		:= SIZEOF(nRevision),
	bDone			=> ,
	bBusy			=> ,
	bError			=> ,
	nErrID			=> ,
	nProcessedLen	=> );

CASE _iRevision OF

	0: (* idle *)
		IF _AdsConn.bDone THEN
			IF stAdsConn.bValid THEN
				_iRevision := 1;
			END_IF
		END_IF
		_ReadRevisionProp.bExecute := FALSE;

	1: (* read property *)
		IF		_ReadRevisionProp.bExecute
			AND	(NOT _ReadRevisionProp.bBusy)
		THEN
			IF _ReadRevisionProp.bError THEN
				nErrorId := BACnet_ERR_REVISION_READ;
			END_IF
			_ReadRevisionProp.bExecute := FALSE;
			_iRevision := 0;
		ELSE
			_ReadRevisionProp.bExecute := TRUE;
		END_IF

END_CASE


(* Handle persistent data backup *)
_nPersistentState := _ePersistentState;
_ReadPersistentProp(
	BACnetDevicePort:= stAdsConn.nAmsPort,
	bExecute		:= ,
	sNetId			:= stAdsConn.sAmsNetId,
	ObjectType		:= BACnetObjectType_Device,
	PropertyID		:= 516,
	DataType		:= BACnetDataType_PersistentDataState,
	ObjectInstance	:= F_BACnet_GetObjInstance(_ObjectId),
	ptrValue		:= ADR(_nPersistentState),
	nLenValue		:= SIZEOF(_nPersistentState),
	bDone			=> ,
	bBusy			=> ,
	bError			=> ,
	nErrID			=> ,
	nProcessedLen	=> );

_WritePersistentProp(
	BACnetDevicePort:= stAdsConn.nAmsPort,
	bExecute		:= ,
	sNetId			:= stAdsConn.sAmsNetId,
	ObjectType		:= BACnetObjectType_Device,
	PropertyID		:= 516,
	Priority		:= ,
	DataType		:= BACnetDataType_PersistentDataState,
	ObjectInstance	:= F_BACnet_GetObjInstance(_ObjectId),
	ptrValue		:= ADR(_nPersistentState),
	nLenValue		:= SIZEOF(_nPersistentState),
	bDone			=> ,
	bBusy			=> ,
	bError			=> ,
	nErrID			=> );
_ePersistentState := UDINT_TO_UINT(_nPersistentState AND 16#0000FFFF);

CASE _iPersis OF
	0: (* idle *)
		IF		bWritePersis
			AND	(NOT bBackupActive)
			AND	(eSystemStatus <> BACnetDeviceStatus_BackupInProgress)
			AND	(nErrorId = BACnet_ERR_NO_ERROR)
		THEN
			IF stAdsConn.bValid THEN
				_iPersis := 1;
			ELSE
				nErrorId := BACnet_ERR_INVALID_ADS_CONN;
			END_IF
		END_IF
		_ReadPersistentProp.bExecute := FALSE;
		_WritePersistentProp.bExecute := FALSE;
		_bPersisWritten := FALSE;

	1: (* read persistent state machine *)
		IF _ReadPersistentProp.bExecute THEN
			IF _ReadPersistentProp.bError THEN
				_iPersis := 100;
				nErrorId := BACnet_ERR_PERSISTENT_WRITE;
				_ReadPersistentProp.bExecute := FALSE;
			ELSIF (NOT _ReadPersistentProp.bBusy) THEN
				_iPersis := 2;
				_ReadPersistentProp.bExecute := FALSE;
			END_IF
		ELSE
			_ReadPersistentProp.bExecute := TRUE;
		END_IF

	2: (* check state *)
		_tonPersisTimeout.IN := FALSE;
		_tonPersisPoll.IN := FALSE;

		IF _tonPersisPoll.Q THEN
			(* rescan state machine *)
			_iPersis := 1;

		ELSIF _tonPersisTimeout.Q THEN
			(* timeout *)
			_iPersis := 100;
			nErrorId := BACnet_ERR_PERSISTENT_WRITE;

		ELSIF (_ePersistentState = BACnetPersistentData_Disabled) THEN
			_iPersis := 10;

		ELSIF	(_ePersistentState = BACnetPersistentData_Initialize)
			OR	(_ePersistentState >= BACnetPersistentData_Write)
		THEN
			(* wait on idle state *)
			_tonPersisTimeout.IN := TRUE;
			_tonPersisPoll.IN := TRUE;

		ELSIF (_ePersistentState = BACnetPersistentData_NoChange) THEN
			(* start writing PLC *)
			_iPersis := 10;

		ELSIF (_ePersistentState = BACnetPersistentData_Ready) THEN
			IF _bPersisWritten THEN
				(* start writing PLC *)
				_iPersis := 10;
			ELSE
				(* start writing BACnet *)
				_iPersis := 3;
			END_IF

		ELSE
			(* wrong state *)
			_iPersis := 100;
			nErrorId := BACnet_ERR_PERSISTENT_WRITE;
		END_IF
		(* call timer *)
		_tonPersisTimeout(PT:= t#60s, Q=> , ET=> );
		_tonPersisPoll(PT:= t#2s, Q=> , ET=> );

	3: (* write BACnet persistent data *)
		IF _WritePersistentProp.bExecute THEN
			IF _WritePersistentProp.bError THEN
				nErrorId := BACnet_ERR_PERSISTENT_WRITE;
				_iPersis := 100;
				_WritePersistentProp.bExecute := FALSE;
			ELSIF (NOT _WritePersistentProp.bBusy) THEN
				_iPersis := 10; (* start writing PLC *)
				_WritePersistentProp.bExecute := FALSE;
				_bPersisWritten := TRUE;
			END_IF
		ELSE
			_WritePersistentProp.bExecute := TRUE;
			_ePersistentState := BACnetPersistentData_Write;
		END_IF

	10: (* write PLC persistent data *)
		IF _fbWritePersistent.START THEN
			IF _fbWritePersistent.ERR THEN
				(* Aborted *)
				nErrorId := BACnet_ERR_PERSISTENT_PLC_WRITE;
				_iPersis := 100;
				_fbWritePersistent.START := FALSE;
			ELSIF (NOT _fbWritePersistent.BUSY) THEN
				(* Finished *)
				_iPersis := 100;
				_fbWritePersistent.START := FALSE;
			END_IF
		ELSE
			_fbWritePersistent.START := TRUE;
		END_IF

	100:
		IF (NOT bWritePersis) THEN
			_iPersis := 0;
		END_IF

END_CASE

(* control *)
(* Disable write-on-change *)
_ServerControl.2	:= bDisableWOC;
(* PLC running - process data valid *)
_ServerControl.11	:=	(NOT _bHasStarted)
					AND	bOperational;

(* state *)
bWritePersisActive := (_iPersis > 0) AND (_iPersis < 100);
bBackupActive := (eSystemStatus = BACnetDeviceStatus_BackupInProgress);
bOperational :=	(_BACnetAdapter^.eAdapterStatus > BACnetAdapterStatus_Init);
bWOCDisabled := (_ServerStatus AND 16#0004) = 16#0004;
_pLocalDate := ADR(_LocalDate);
_pLocalTime := ADR(_LocalTime);
dtLocalTime.stDate := _pLocalDate^;
dtLocalTime.stTime := _pLocalTime^;

(* update counter *)
IF (_nUpdateCount = 0) AND _bHasStarted THEN
	bFirstCycle := TRUE;
ELSE
	bFirstCycle := FALSE;
END_IF
_bHasStarted := FALSE;
_nUpdateCount := _nUpdateCount + 1;
bError := (nErrorId <> BACnet_ERR_NO_ERROR);
END_FUNCTION_BLOCK

(* POU FB_BACnet_Adapter, ST *)
FUNCTION_BLOCK FB_BACnet_Adapter
VAR_INPUT
END_VAR
VAR_OUTPUT
	eAdapterStatus		: E_BACNETADAPTERSTATUS;
	bEthLinkOk			: BOOL;
	bGatewayOk			: BOOL;
	sAmsNetId			: T_AmsNetId;
	bFirstCycle			: BOOL;
	bError				: BOOL;
	nErrorId			: UINT;
END_VAR
VAR
	_DeviceStatus	AT%I*: WORD; (* ~(BACnet_DeviceStatus : : ) *)
	_AmsNetId		AT%I*: ARRAY[0..5] OF BYTE; (* ~(BACnet_AmsNetId : : ) *)
	_bHasStarted	: BOOL := TRUE;
	_nUpdateCount	: UDINT := 0;
END_VAR
(* reset error ID *)
nErrorId	:= BACnet_ERR_NO_ERROR;
bError		:= FALSE;

(* update bacnet adapter pointer *)
pBACnet_Adapter := ADRINST();

(* convert _DeviceStatus to enumeration *)
eAdapterStatus := SHR((_DeviceStatus AND 16#FF00), 8);

(* update netid *)
UpdateNetID();

(* states *)
bEthLinkOk := (NOT _DeviceStatus.0);
bGatewayOk := (eAdapterStatus = BACnetAdapterStatus_Complete) AND bEthLinkOk;

(* update counter *)
IF (_nUpdateCount = 0) AND _bHasStarted THEN
	bFirstCycle := TRUE;
	_bHasStarted := FALSE;
ELSE
	bFirstCycle := FALSE;
END_IF
_nUpdateCount := _nUpdateCount +1;
END_FUNCTION_BLOCK
ACTION UpdateNetID:
(* read NetId and convert to string *)
sAmsNetId := F_CreateAmsNetId(_AmsNetId);
(* check if it plausible *)
IF sAmsNetId = '0.0.0.0.0.0' THEN
	(* NetId not OK, return with error *)
	bError := TRUE;
	nErrorId := BACnet_ERR_NO_VALID_NET_ID;
	sAmsNetId := '';
END_IF
END_ACTION

(* POU FB_BACnet_WriteProp, ST *)
FUNCTION_BLOCK FB_BACnet_WriteProp
VAR_INPUT
	BACnetDevicePort	: UINT := 16#FFFF;
	bExecute			: BOOL;
	sNetId				: T_AmsNetId;
	ObjectType			: E_BACNETOBJECTTYPE;
	PropertyID			: E_BACNETPROPERTYIDENTIFIER;
	Priority			: E_BACNETPRIORITY;
	DataType			: E_BACNETDATATYPES;
	ObjectInstance		: UDINT;
	ptrValue			: POINTER TO BYTE;
	nLenValue			: UDINT; (* byte size of value (SIZEOF) *)
END_VAR
VAR_OUTPUT
	bDone				: BOOL;
	bBusy				: BOOL;
	bError				: BOOL;
	nErrID				: UDINT;
END_VAR
VAR
	_Write				: ADSWRITE;
	_rtrigStart			: R_TRIG;
	_len_data			: UDINT;
	_nPrio 				: UDINT;
	_ptrDWORD			: POINTER TO DWORD;
	_ptrREAL			: POINTER TO REAL;
	_ptrBYTE			: POINTER TO BYTE;
	_dataPointer		: POINTER TO BYTE;
	_dwordVal			: DWORD;
END_VAR
(* catch the start flag *)
	_rtrigStart(Clk:=bExecute);

(* prepare *)
	IF _rtrigStart.Q AND (NOT bBusy) THEN
		_Write(WRITE := FALSE);
		bDone := FALSE;
		bBusy := TRUE;
		bError := FALSE;
		nErrId := 0;
		_nPrio := SHL(INT_TO_UDINT(Priority), 26);
		_len_data := nLenValue; (* in default, take the user given length *)
		_dataPointer := ptrValue;
		CASE DataType OF
			BACnetDataType_Null 				: _len_data := 0; (* set length to zero *)
			BACnetDataType_Bool 				: _len_data := _len_data; (* 1 *)
			BACnetDataType_CharacterStringExt	: _len_data := _len_data; (* 2 *)

			BACnetDataType_UnsignedInteger,
			BACnetDataType_SignedInteger 		: _len_data := MIN(_len_data, 4); (* 4 *)
				IF (_len_data >= 4) THEN
					(* source data type bigger/equal 4 byte --> OK, take first 4 byte *)
					_ptrDWORD := ptrValue;
				ELSE
					(* upgrade data type from less 4 byte to fully double word *)
					_dwordVal := 0;
					_ptrDWORD := ADR(_dwordVal);
					MEMCPY(destAddr:=_ptrDWORD, srcAddr:=ptrValue, n:=_len_data);
					_dataPointer := _ptrDWORD; (* from here on, point to the internal data source *)
					_len_data := SIZEOF(_dwordVal); (* increase size to internal data type length *)
				END_IF
				(* make some plausibility checks *)
				IF	(		ObjectType = BACnetObjectType_MultiStateInput
						OR	ObjectType = BACnetObjectType_MultiStateOutput
						OR	ObjectType = BACnetObjectType_MultiStateValue
					)
				THEN
					IF _ptrDWORD^ = 0 THEN
						(* set data type and data length to NULL operation *)
						_len_data := 0;
					END_IF
				END_IF

			BACnetDataType_Real 				: _len_data := _len_data; (* 4 *)
				_ptrREAL := ptrValue;
				IF (NOT F_BACnet_IsFinite(_ptrREAL^)) THEN
					(* set data type and data length to NULL operation *)
					_len_data := 0;
				END_IF

			BACnetDataType_Double 				: _len_data := _len_data; (* 8 *)
			BACnetDataType_OctetString 			: _len_data := _len_data; (* 8 *)
			BACnetDataType_Enumerated 			: _len_data := _len_data; (* 8 *)
			BACnetDataType_LimitEnable			: _len_data := _len_data; (* 4 *)
			BACnetDataType_BitString 			: _len_data := _len_data; (* 11 *)

			BACnetDataType_BinaryPV				: _len_data := MIN(_len_data, 1); (* 1 *)
				_ptrByte := ptrValue;
				IF		_len_data <= 0
					OR	_ptrByte^ >= 2
				THEN
					_len_data := 0;
				END_IF
		END_CASE
	ELSIF (NOT bExecute) THEN
		bDone := FALSE;
	END_IF

(* execute *)
	IF bBusy THEN
		_Write(	NETID:= sNetId,
				PORT:= BACnetDevicePort,
				IDXGRP:=16#80000000 + INT_TO_UDINT(PropertyID) + _nPrio,
				IDXOFFS:= F_BACnet_GetObjId(ObjectType, ObjectInstance),
				LEN:= _len_data,
				SRCADDR:= _dataPointer,
				WRITE:= TRUE,
				TMOUT:= BACnet_ADSTimeOut);
		IF NOT _Write.Busy THEN
			IF _Write.Err THEN
				nErrID := _Write.ErrId;
				bError := TRUE;
			END_IF
			_Write(WRITE := FALSE);
			bBusy := FALSE;
			bDone := NOT bError;
		END_IF
	END_IF
END_FUNCTION_BLOCK

(* POU FB_BACnet_ReadProp, ST *)
FUNCTION_BLOCK FB_BACnet_ReadProp
VAR_INPUT
	BACnetDevicePort	: UINT := 16#FFFF;
	bExecute			: BOOL;
	sNetId				: T_AmsNetId;
	ObjectType			: E_BACNETOBJECTTYPE;
	PropertyID			: E_BACNETPROPERTYIDENTIFIER;
	DataType			: E_BACNETDATATYPES;
	ObjectInstance		: DINT;
	ptrValue			: POINTER TO BYTE;
	nLenValue			: UDINT; (* byte size of value (SIZEOF) *)
END_VAR
VAR_OUTPUT
	bDone				: BOOL;
	bBusy				: BOOL;
	bError				: BOOL;
	nErrID				: UDINT;
	nProcessedLen		: UDINT; (* the received data length (can be different to given length) *)
END_VAR
VAR
	_Read				: FW_AdsRead;
	_rtrigStart			: R_TRIG;
	_len_data			: UDINT;
END_VAR
(* catch the start flag *)
	_rtrigStart(Clk:=bExecute);

(* prepare *)
	IF _rtrigStart.Q AND (NOT bBusy) THEN
		_Read(bExecute := FALSE);
		bDone := FALSE;
		bBusy := TRUE;
		bError := FALSE;
		nErrId := 0;
		nProcessedLen := 0;
		(* in default, take the user given length *)
		_len_data := nLenValue;
		(* set index group for read property access *)
		_Read.nIdxGrp := 16#80000000 + INT_TO_UDINT(PropertyID);
		(* handle special data type things *)
		CASE DataType OF
			BACnetDataType_Null 				: _len_data := 0; (* set length to zero *)
			BACnetDataType_Bool 				: _len_data := _len_data; (* 1 *)
			BACnetDataType_CharacterStringExt	: _len_data := _len_data; (* 2 *)
			BACnetDataType_UnsignedInteger 		: _len_data := _len_data; (* 4 *)
			BACnetDataType_SignedInteger 		: _len_data := _len_data; (* 4 *)
			BACnetDataType_Real 				: _len_data := _len_data; (* 4 *)
			BACnetDataType_Double 				: _len_data := _len_data; (* 8 *)
			BACnetDataType_OctetString 			: _len_data := _len_data; (* 8 *)
			BACnetDataType_Enumerated 			: _len_data := _len_data; (* 8 *)
			BACnetDataType_LimitEnable			: _len_data := _len_data; (* 4 *)
			BACnetDataType_BitString 			: _len_data := _len_data; (* 11 *)
			BACnetDataType_LogRecordList:
				_len_data := _len_data; (* n *)
				_Read.nIdxGrp := _Read.nIdxGrp + 16#03800000; (* read range *)
		END_CASE;
	ELSIF (NOT bExecute) THEN
		bDone := FALSE;
	END_IF


(* execute *)
	IF bBusy THEN
		_Read(
			sNetId		:= sNetId,
			nPort		:= BACnetDevicePort,
			nIdxGrp		:= , (* see above *)
			nIdxOffs	:= F_BACnet_GetObjId(ObjectType, ObjectInstance),
			cbReadLen	:= _len_data,
			pReadBuff	:= ptrValue,
			bExecute	:= TRUE,
			tTimeout	:= BACnet_ADSTimeOut,
			bBusy		=> ,
			bError		=> ,
			nErrId		=> ,
			cbRead		=> );
		IF (NOT _Read.bBusy) THEN
			IF _Read.bError THEN
				nErrID := _Read.nErrId;
				bError := TRUE;
				nProcessedLen := 0;
			ELSE
				(* success *)
				nProcessedLen := _Read.cbRead;
				IF (_Read.cbRead < nLenValue) THEN
					(* fill unused part of buffer with zero *)
					MEMSET(destAddr:=(ptrValue+_Read.cbRead), fillByte:=0, n:=(nLenValue-_Read.cbRead));
				END_IF
			END_IF
			_Read(bExecute := FALSE);
			bBusy := FALSE;
			bDone := NOT bError;
		END_IF;
	END_IF
END_FUNCTION_BLOCK

(* POU FB_BACnet_Accumulator_EX, ST *)
FUNCTION_BLOCK FB_BACnet_Accumulator_EX
VAR_INPUT
	nPV					: UDINT; (* number for present_value *)
END_VAR
VAR_IN_OUT
	Device				: FB_BACnet_Device;
END_VAR
VAR_OUTPUT
	bReady				: BOOL;
	nPresentValue		: UDINT;
	nMaxPV				: UDINT;
	bOverridden			: BOOL;
	bOutOfService		: BOOL;
	bFault				: BOOL;
	bInAlarm			: BOOL;
	bOverRange			: BOOL;
	bUnderRange			: BOOL;
	bNoSensor			: BOOL;
	bOpenLoop			: BOOL;
	bCommFailure		: BOOL;
	bShortedLoop		: BOOL;
	bOtherFault			: BOOL;
	eEventState			: E_BACNETEVENTSTATE;
	tObjectID			: T_BACnet_ObjectIdentifier := 16#FFFFFFFF;
	bError				: BOOL;
	nErrorId			: UINT;
END_VAR
VAR
	_PresentValueIn AT%I*:UDINT;	(* ~(BACnet_PresentValue	:		: )
										(BACnet_ObjectType		: ACC	: )	*)
    _PresentValueOut AT%Q*:UDINT;	(* ~(BACnet_PresentValue	:		: )	*)
	_MaxPresValue AT%I*:UDINT;		(* ~(BACnet_MaxPresValue	:		: writeprotect) *)
	_ObjectId AT%I*: DWORD;			(* ~(BACnet_ObjectIdentifier:		: LINK) *)
	_StatusFlags AT%I*:WORD;		(* ~(BACnet_StatusFlags		:		: )	*)
	_EventState AT%I*: WORD; 		(* ~(BACnet_EventState 		:		: )	*)
	_Reliability AT%I*: WORD; 		(* ~(BACnet_Reliability 	:		: )	*)
	_nUpdateCount : UDINT := 0;
	_StatusFlagsBits : ST_BACnet_StatusFlags;
END_VAR
(* update client device *)
IF (Device._nUpdateCount = _nUpdateCount) THEN
	Device();
END_IF
(* remind current number of update counter *)
_nUpdateCount := Device._nUpdateCount;

(* check object type *)
IF (F_BACnet_GetObjType(_ObjectId) <> BACnetObjectType_Accumulator) THEN
	(* wrong mapping / invalid object ID *)
	IF _ObjectId = 0 THEN
		nErrorId := BACnet_ERR_WRONG_MAPPING;
	ELSE
		nErrorId := BACnet_ERR_INVALID_OBJECTID;
	END_IF
	bReady := FALSE;

ELSIF _StatusFlags < 4 THEN
	(* mapping seems to be wrong (bit string for status flags must be 4 in minimum) *)
	nErrorId := BACnet_ERR_WRONG_MAPPING;

ELSIF Device.bOperational THEN
	(* clear error flag *)
	nErrorId := BACnet_ERR_NO_ERROR;
	bReady := TRUE;
	(* copy present value *)
	nPresentValue 		:= _PresentValueIn;
	_PresentValueOut	:= nPV;
	nMaxPV				:= _MaxPresValue;

	(* build bit states *)
	_StatusFlagsBits	:= F_BACnet_StatusFlags(_StatusFlags);

	(* copy states to output *)
	bOverridden := _StatusFlagsBits.overridden;
	bOutOfService := _StatusFlagsBits.out_of_service;
	bFault := _StatusFlagsBits.fault;
	bInAlarm := _StatusFlagsBits.in_alarm;
	bOverRange := (_Reliability = BACnetReliability_over_range);
	bUnderRange := (_Reliability = BACnetReliability_under_range);
	bNoSensor := (_Reliability = BACnetReliability_no_sensor);
	bOpenLoop := (_Reliability = BACnetReliability_open_loop);
	bCommFailure := (_Reliability = BACnetReliability_communication_failure);
	bShortedLoop := (_Reliability = BACnetReliability_shorted_loop);
	bOtherFault := (_Reliability = BACnetReliability_unreliable_other);
	tObjectID := _ObjectId;

	(* convert enumeration *)
	eEventState := _EventState;
ELSE
	bReady := FALSE;
	(* and set error ID *)
	nErrorId := BACnet_ERR_OPERATIONAL;
END_IF

(* set error flag *)
bError := (nErrorId <> BACnet_ERR_NO_ERROR);
END_FUNCTION_BLOCK

(* POU FB_BACnet_Accumulator_R6, ST *)
FUNCTION_BLOCK FB_BACnet_Accumulator_R6
VAR_INPUT
	nPV					: UDINT; (* number for present_value *)
END_VAR
VAR_IN_OUT
	Device				: FB_BACnet_Device;
END_VAR
VAR_OUTPUT
	bReady				: BOOL;
	nPresentValue		: UDINT;
	bOverridden			: BOOL;
	bOutOfService		: BOOL;
	bFault				: BOOL;
	bInAlarm			: BOOL;
	bError				: BOOL;
	nErrorId			: UINT;
END_VAR
VAR
	_PresentValueIn AT%I*:UDINT;	(* ~(BACnet_PresentValue	:		: )
										(BACnet_MaxPresValue	:		: writeprotect,nolink)
										(BACnet_ObjectType		: ACC	: )	*)
    _PresentValueOut AT%Q*:UDINT;	(* ~(BACnet_PresentValue	:		: )	*)
	_StatusFlags AT%I*:WORD;		(* ~(BACnet_StatusFlags		:		: )	*)
	_StatusFlagsBits : ST_BACnet_StatusFlags;

	_nUpdateCount : UDINT := 0;
END_VAR
(* update device *)
IF (Device._nUpdateCount = _nUpdateCount) THEN
	Device();
END_IF
(* remind current number of update counter *)
_nUpdateCount := Device._nUpdateCount;

IF _StatusFlags < 4 THEN
	(* mapping seems to be wrong (bit string for status flags must be 4 in minimum) *)
	nErrorId := BACnet_ERR_WRONG_MAPPING;

ELSIF Device.bOperational THEN
	(* clear error flag *)
	nErrorId := BACnet_ERR_NO_ERROR;
	bReady := TRUE;
	(* copy present value *)
	nPresentValue 		:= _PresentValueIn;
	_PresentValueOut	:= nPV;

	(* build bit states *)
	_StatusFlagsBits	:= F_BACnet_StatusFlags(_StatusFlags);

	(* copy states to output *)
	bOverridden := _StatusFlagsBits.overridden;
	bOutOfService := _StatusFlagsBits.out_of_service;
	bFault := _StatusFlagsBits.fault;
	bInAlarm := _StatusFlagsBits.in_alarm;
ELSE
	bReady := FALSE;
	(* and set error ID *)
	nErrorId := BACnet_ERR_OPERATIONAL;
END_IF

(* set error flag *)
bError := (nErrorId <> BACnet_ERR_NO_ERROR);
END_FUNCTION_BLOCK

(* POU FB_BACnet_Accumulator_RAW, ST *)
FUNCTION_BLOCK FB_BACnet_Accumulator_RAW
VAR_INPUT
	nRawIn				AT%Q*: UINT; (* ~(BACnet_RawIoAccumulatorUnsignedValue : : ) *)
	bNoSensor			: BOOL;
	bOverRange			: BOOL;
	bUnderRange			: BOOL;
	bOpenLoop			: BOOL;
	bShortedLoop		: BOOL;
	bCommFailure		: BOOL;
	bOtherFault			: BOOL;
END_VAR
VAR_IN_OUT
	Device				: FB_BACnet_Device;
END_VAR
VAR_OUTPUT
	bReady				: BOOL;
	nPresentValue		: UDINT;
	bOverridden			: BOOL;
	bOutOfService		: BOOL;
	bFault				: BOOL;
	bInAlarm			: BOOL;
	bError				: BOOL;
	nErrorId			: UINT;
END_VAR
VAR
	_PresentValueIn AT%I*:UDINT;	(* ~(BACnet_PresentValue	:		: )
										(BACnet_MaxPresValue	:		: writeprotect,nolink)
										(BACnet_ObjectType		: ACC	: )	*)
	_ObjectId AT%I*: DWORD;			(* ~(BACnet_ObjectIdentifier:		: LINK) *)
	_StatusFlags AT%I*:WORD;		(* ~(BACnet_StatusFlags		:		: )	*)
	_ReliabilityIn AT%I*: WORD;		(* ~(BACnet_Reliability 	:		: )	*)
	_ReliabilityOut AT%Q*: WORD := BACnetReliability_no_fault_detected;(* ~(BACnet_Reliability 	:		: )	*)
	_StatusFlagsBits : ST_BACnet_StatusFlags;

	_nUpdateCount : UDINT := 0;
END_VAR
(* update device *)
IF Device._nUpdateCount = _nUpdateCount THEN
	Device();
END_IF
(* remind current number of update counter *)
_nUpdateCount := Device._nUpdateCount;

(* handle raw error *)
IF bNoSensor THEN
	_ReliabilityOut := BACnetReliability_no_sensor;
ELSIF bOverRange THEN
	_ReliabilityOut := BACnetReliability_over_range;
ELSIF bUnderRange THEN
	_ReliabilityOut := BACnetReliability_under_range;
ELSIF bOpenLoop THEN
	_ReliabilityOut := BACnetReliability_open_loop;
ELSIF bShortedLoop THEN
	_ReliabilityOut := BACnetReliability_shorted_loop;
ELSIF bCommFailure THEN
	_ReliabilityOut := BACnetReliability_communication_failure;
ELSIF bOtherFault THEN
	_ReliabilityOut := BACnetReliability_unreliable_other;
ELSE
	_ReliabilityOut := BACnetReliability_no_fault_detected;
END_IF

IF _StatusFlags < 4 THEN
	(* mapping seems to be wrong (bit string for status flags must be 4 in minimum) *)
	nErrorId := BACnet_ERR_WRONG_MAPPING;

ELSIF Device.bOperational THEN
	(* clear error flag *)
	nErrorId := BACnet_ERR_NO_ERROR;
	bReady := TRUE;
	(* copy present value *)
	nPresentValue 		:= _PresentValueIn;

	(* build bit states *)
	_StatusFlagsBits	:= F_BACnet_StatusFlags(_StatusFlags);

	(* copy states to output *)
	bOverridden := _StatusFlagsBits.overridden;
	bOutOfService := _StatusFlagsBits.out_of_service;
	bFault := _StatusFlagsBits.fault;
	bInAlarm := _StatusFlagsBits.in_alarm;
ELSE
	bReady := FALSE;
	(* and set error ID *)
	nErrorId := BACnet_ERR_OPERATIONAL;
END_IF

(* set error flag *)
bError := (nErrorId <> BACnet_ERR_NO_ERROR);
END_FUNCTION_BLOCK

(* POU FB_BACnet_Accumulator_RAW_R6, ST *)
FUNCTION_BLOCK FB_BACnet_Accumulator_RAW_R6
VAR_INPUT
	nPV					: UDINT; (* number for present_value *)
	nReliability		: WORD;
	bOutOfServiceOut	: BOOL;
END_VAR
VAR_IN_OUT
	Device				: FB_BACnet_Device;
END_VAR
VAR_OUTPUT
	bReady				: BOOL;
	nPresentValue		: UDINT;
	nMaxPV				: UDINT;
	bOverridden			: BOOL;
	bOutOfService		: BOOL;
	bFault				: BOOL;
	bInAlarm			: BOOL;
	bOverRange			: BOOL;
	bUnderRange			: BOOL;
	bNoSensor			: BOOL;
	bOpenLoop			: BOOL;
	bShortedLoop		: BOOL;
	bOtherFault			: BOOL;
	eEventState			: E_BACNETEVENTSTATE;
	bError				: BOOL;
	nErrorId			: UINT;
END_VAR
VAR
	_PresentValueIn AT%I*:UDINT;	(* ~(BACnet_PresentValue	:		: )
										(BACnet_ObjectType		: ACC	: )	*)
    _PresentValueOut AT%Q*:UDINT;	(* ~(BACnet_PresentValue	:		: )	*)
	_MaxPresValue AT%I*:UDINT;		(* ~(BACnet_MaxPresValue	:		: writeprotect) *)
	_StatusFlags AT%I*:WORD;		(* ~(BACnet_StatusFlags		:		: )	*)
	_EventState AT%I*: WORD; 		(* ~(BACnet_EventState 		:		: )	*)
	_Reliability AT%I*: WORD; 		(* ~(BACnet_Reliability 	:		: )	*)
	_StatusFlagsOut AT%Q*:WORD;		(* ~(BACnet_StatusFlags		:		: )	*)
	_EventStateOut AT%Q*: WORD;		(* ~(BACnet_EventState 		:		: )	*)
	_ReliabilityOut AT%Q*: WORD;	(* ~(BACnet_Reliability 	:		: )	*)
	_OutOfServiceOut AT%Q*: BOOL;	(* ~(BACnet_OutOfService	:		: writeprotect) *)
	_StatusFlagsBits : ST_BACnet_StatusFlags;
	_StatusFlagsOutBits : ST_BACnet_StatusFlags;
	_nUpdateCount : UDINT := 0;
END_VAR
(* update client device *)
IF (Device._nUpdateCount = _nUpdateCount) THEN
	Device();
END_IF
(* remind current number of update counter *)
_nUpdateCount := Device._nUpdateCount;

(* copy reliability and out of service flags *)
_ReliabilityOut		:= nReliability;
_OutOfServiceOut	:= bOutOfServiceOut;

IF _StatusFlags < 4 THEN
	(* mapping seems to be wrong (bit string for status flags must be 4 in minimum) *)
	nErrorId := BACnet_ERR_WRONG_MAPPING;

ELSIF Device.bOperational THEN
	(* clear error flag *)
	nErrorId := BACnet_ERR_NO_ERROR;
	bReady := TRUE;
	(* copy present value *)
	nPresentValue 		:= _PresentValueIn;
	_PresentValueOut	:= nPV;
	nMaxPV				:= _MaxPresValue;

	(* build bit states *)
	_StatusFlagsBits	:= F_BACnet_StatusFlags(_StatusFlags);

	(* copy states to output *)
	bOverridden := _StatusFlagsBits.overridden;
	bOutOfService := _StatusFlagsBits.out_of_service;
	bFault := _StatusFlagsBits.fault;
	bInAlarm := _StatusFlagsBits.in_alarm;
	bOverRange := (_Reliability = BACnetReliability_over_range);
	bUnderRange := (_Reliability = BACnetReliability_under_range);
	bNoSensor := (_Reliability = BACnetReliability_no_sensor);
	bOpenLoop := (_Reliability = BACnetReliability_open_loop);
	bShortedLoop := (_Reliability = BACnetReliability_shorted_loop);
	bOtherFault := (_Reliability = BACnetReliability_unreliable_other);

	(* convert enumeration *)
	eEventState := _EventState;
ELSE
	bReady := FALSE;
	(* and set error ID *)
	nErrorId := BACnet_ERR_OPERATIONAL;
END_IF

(* set status flags depending on reliability *)
IF _ReliabilityOut = BACnetReliability_no_fault_detected THEN
	_StatusFlagsOutBits.fault := FALSE;
	_StatusFlagsOutBits.in_alarm := FALSE;
	_EventStateOut := 0;
ELSE
	_StatusFlagsOutBits.fault := TRUE;
	_StatusFlagsOutBits.in_alarm := TRUE;
	_EventStateOut := 1;
END_IF

_StatusFlagsOutBits.out_of_service := _OutOfServiceOut;
_StatusFlagsOut	:= F_BACnet_GetStatusFlagsData(_StatusFlagsOutBits);

(* set error flag *)
bError := (nErrorId <> BACnet_ERR_NO_ERROR);
END_FUNCTION_BLOCK

(* POU FB_BACnet_AnalogInput, ST *)
FUNCTION_BLOCK FB_BACnet_AnalogInput
VAR_IN_OUT
	Device	: FB_BACnet_Device;
END_VAR
VAR_OUTPUT
	bReady			: BOOL;
	fPresentValue	: REAL;
	bOverridden		: BOOL;
	bOutOfService	: BOOL;
	bFault			: BOOL;
	bInAlarm		: BOOL;
	bError			: BOOL;
	nErrorId		: UINT;
END_VAR
VAR
	_PresentValue AT%I*: REAL; 		(* ~(BACnet_PresentValue 	:		: )
								   		(BACnet_ObjectType 		: AI	: )	*)
	_StatusFlags AT%I*: WORD; 		(* ~(BACnet_StatusFlags 	:		: )	*)
	_StatusFlagsBits : ST_BACnet_StatusFlags;
	_nUpdateCount : UDINT := 0;
END_VAR
(* update server device *)
IF (Device._nUpdateCount = _nUpdateCount) THEN
	Device();
END_IF
(* remind current number of update counter *)
_nUpdateCount := Device._nUpdateCount;

(* check BitString format of StatusFlags --> if StatusFlags are less than 4, object isn't linked correctly *)
IF (_StatusFlags < 4) THEN
	(* wrong mapping *)
	nErrorId := BACnet_ERR_WRONG_MAPPING;
	bReady := FALSE;

ELSIF Device.bOperational THEN
	(* ready state *)
	bReady := TRUE;
	nErrorId := BACnet_ERR_NO_ERROR;

	(* present value *)
	fPresentValue := _PresentValue;

	(* build bit states *)
	_StatusFlagsBits := F_BACnet_StatusFlags(_StatusFlags);

	(* copy states to output *)
	bOverridden := _StatusFlagsBits.overridden;
	bOutOfService := _StatusFlagsBits.out_of_service;
	bFault := _StatusFlagsBits.fault;
	bInAlarm := _StatusFlagsBits.in_alarm;
ELSE
	(* server device not ready, reset local ready also *)
	bReady := FALSE;
	nErrorId := BACnet_ERR_OPERATIONAL;
END_IF
(* set error flag *)
bError := (nErrorId <> BACnet_ERR_NO_ERROR);
END_FUNCTION_BLOCK

(* POU FB_BACnet_AnalogInput_EX, ST *)
FUNCTION_BLOCK FB_BACnet_AnalogInput_EX
VAR_IN_OUT
	Device				: FB_BACnet_Device;
END_VAR
VAR_OUTPUT
	bReady				: BOOL;
	fPresentValue		: REAL;
	bOverridden			: BOOL;
	bOutOfService		: BOOL;
	bFault				: BOOL;
	bInAlarm			: BOOL;
	bOverRange			: BOOL;
	bUnderRange			: BOOL;
	bNoSensor			: BOOL;
	bOpenLoop			: BOOL;
	bShortedLoop		: BOOL;
	bOtherFault			: BOOL;
	eEventState			: E_BACNETEVENTSTATE;
	bAckedTrans_ToOffNormal : BOOL;
	bAckedTrans_ToFault		: BOOL;
	bAckedTrans_ToNormal	: BOOL;
	tObjectID			: T_BACnet_ObjectIdentifier := 16#FFFFFFFF;
	bError				: BOOL;
	nErrorId			: UINT;
END_VAR
VAR
	_PresentValue AT%I*: REAL; 			(* ~(BACnet_PresentValue 	:		: )
								   			(BACnet_ObjectType 		: AI	: )	*)
	_ObjectId AT%I*: DWORD;				(* ~(BACnet_ObjectIdentifier:		: LINK) *)
	_StatusFlags AT%I*: WORD; 			(* ~(BACnet_StatusFlags 	:		: )	*)
	_EventState AT%I*: WORD; 			(* ~(BACnet_EventState 		:		: )	*)
	_Reliability AT%I*: WORD; 			(* ~(BACnet_Reliability 	:		: )	*)
	_AckedTransitions AT%I*:WORD;		(* ~(BACnet_AckedTransitions:		: ) *)
	_AckedTransBits : ST_BACnet_EventTransitionBits;
	_StatusFlagsBits : ST_BACnet_StatusFlags;
	_nUpdateCount : UDINT := 0;
END_VAR
(* update server device *)
IF (Device._nUpdateCount = _nUpdateCount) THEN
	Device();
END_IF
(* remind current number of update counter *)
_nUpdateCount := Device._nUpdateCount;

(* check object type *)
IF (F_BACnet_GetObjType(_ObjectId) <> BACnetObjectType_AnalogInput) THEN
	(* wrong mapping / invalid object ID *)
	IF _ObjectId = 0 THEN
		nErrorId := BACnet_ERR_WRONG_MAPPING;
	ELSE
		nErrorId := BACnet_ERR_INVALID_OBJECTID;
	END_IF
	bReady := FALSE;
	tObjectID := 16#FFFFFFFF;

ELSIF (_StatusFlags < 4) THEN
	(* mapping seems to be wrong (bit string for status flags must be 4 in minimum) *)
	(* wrong mapping *)
	nErrorId := BACnet_ERR_WRONG_MAPPING;
	bReady := FALSE;

ELSIF Device.bOperational THEN
	(* ready state *)
	bReady := TRUE;
	nErrorId := BACnet_ERR_NO_ERROR;

	(* present value *)
	fPresentValue := _PresentValue;

	(* build bit states *)
	_StatusFlagsBits := F_BACnet_StatusFlags(_StatusFlags);
	_AckedTransBits		:= F_BACnet_EventTransitionFlags(_AckedTransitions);

	(* copy states to output *)
	bOverridden := _StatusFlagsBits.overridden;
	bOutOfService := _StatusFlagsBits.out_of_service;
	bFault := _StatusFlagsBits.fault;
	bInAlarm := _StatusFlagsBits.in_alarm;
	bOverRange := (_Reliability = BACnetReliability_over_range);
	bUnderRange := (_Reliability = BACnetReliability_under_range);
	bNoSensor := (_Reliability = BACnetReliability_no_sensor);
	bOpenLoop := (_Reliability = BACnetReliability_open_loop);
	bShortedLoop := (_Reliability = BACnetReliability_shorted_loop);
	bOtherFault := (_Reliability = BACnetReliability_unreliable_other);
	bAckedTrans_ToOffNormal := _AckedTransBits.to_offnormal;
	bAckedTrans_ToFault := _AckedTransBits.to_fault;
	bAckedTrans_ToNormal := _AckedTransBits.to_normal;
	tObjectID := _ObjectId;

	(* convert enumeration *)
	eEventState := _EventState;
ELSE
	(* server device not ready, reset local ready also *)
	bReady := FALSE;
	nErrorId := BACnet_ERR_OPERATIONAL;
END_IF
(* set error flag *)
bError := (nErrorId <> BACnet_ERR_NO_ERROR);
END_FUNCTION_BLOCK

(* POU FB_BACnet_AnalogInput_RAW, ST *)
FUNCTION_BLOCK FB_BACnet_AnalogInput_RAW
VAR_INPUT
	nRawIn			AT%Q*: INT; (* ~(BACnet_RawIoAnalogSignedValue : : ) *)
	bNoSensor		: BOOL;
	bOverRange		: BOOL;
	bUnderRange		: BOOL;
	bOpenLoop		: BOOL;
	bShortedLoop	: BOOL;
	bCommFailure	: BOOL;
	bOtherFault		: BOOL;
END_VAR
VAR_IN_OUT
	Device	: FB_BACnet_Device;
END_VAR
VAR_OUTPUT
	bReady			: BOOL;
	fPresentValue	: REAL;
	bOverridden		: BOOL;
	bOutOfService	: BOOL;
	bFault			: BOOL;
	bInAlarm		: BOOL;
	bAckedTrans_ToOffNormal : BOOL;
	bAckedTrans_ToFault		: BOOL;
	bAckedTrans_ToNormal	: BOOL;
	bError			: BOOL;
	nErrorId		: UINT;
END_VAR
VAR
	_Reliability AT%Q*: WORD := BACnetReliability_no_fault_detected;(* ~(BACnet_Reliability 	:		: )	*)
	_PresentValue AT%I*: REAL; 		(* ~(BACnet_PresentValue 	:		: )
								   		(BACnet_ObjectType 		: AI	: )	*)
	_ObjectId AT%I*: DWORD;			(* ~(BACnet_ObjectIdentifier:		: LINK) *)
	_AckedTransitions AT%I*:WORD;	(* ~(BACnet_AckedTransitions:		: ) *)
	_StatusFlags AT%I*: WORD; 		(* ~(BACnet_StatusFlags 	:		: )	*)
	_AckedTransBits : ST_BACnet_EventTransitionBits;
	_StatusFlagsBits : ST_BACnet_StatusFlags;
	_nUpdateCount : UDINT := 0;
END_VAR
(* update server device *)
IF (Device._nUpdateCount = _nUpdateCount) THEN
	Device();
END_IF
(* remind current number of update counter *)
_nUpdateCount := Device._nUpdateCount;

(* handle raw error *)
IF bNoSensor THEN
	_Reliability := BACnetReliability_no_sensor;
ELSIF bOverRange THEN
	_Reliability := BACnetReliability_over_range;
ELSIF bUnderRange THEN
	_Reliability := BACnetReliability_under_range;
ELSIF bOpenLoop THEN
	_Reliability := BACnetReliability_open_loop;
ELSIF bShortedLoop THEN
	_Reliability := BACnetReliability_shorted_loop;
ELSIF bCommFailure THEN
	_Reliability := BACnetReliability_communication_failure;
ELSIF bOtherFault THEN
	_Reliability := BACnetReliability_unreliable_other;
ELSE
	_Reliability := BACnetReliability_no_fault_detected;
END_IF

(* check BitString format of StatusFlags --> if StatusFlags are less than 4, object isn't linked correctly *)
IF (_StatusFlags < 4) THEN
	(* wrong mapping *)
	nErrorId := BACnet_ERR_WRONG_MAPPING;
	bReady := FALSE;

ELSIF Device.bOperational THEN
	(* ready state *)
	bReady := TRUE;
	nErrorId := BACnet_ERR_NO_ERROR;

	(* present value *)
	fPresentValue := _PresentValue;

	(* build bit states *)
	_StatusFlagsBits := F_BACnet_StatusFlags(_StatusFlags);
	_AckedTransBits		:= F_BACnet_EventTransitionFlags(_AckedTransitions);

	(* copy states to output *)
	bOverridden := _StatusFlagsBits.overridden;
	bOutOfService := _StatusFlagsBits.out_of_service;
	bFault := _StatusFlagsBits.fault;
	bInAlarm := _StatusFlagsBits.in_alarm;
	bAckedTrans_ToOffNormal := _AckedTransBits.to_offnormal;
	bAckedTrans_ToFault := _AckedTransBits.to_fault;
	bAckedTrans_ToNormal := _AckedTransBits.to_normal;
ELSE
	(* server device not ready, reset local ready also *)
	bReady := FALSE;
	nErrorId := BACnet_ERR_OPERATIONAL;
END_IF
(* set error flag *)
bError := (nErrorId <> BACnet_ERR_NO_ERROR);
END_FUNCTION_BLOCK

(* POU FB_BACnet_AnalogOutput, ST *)
FUNCTION_BLOCK FB_BACnet_AnalogOutput
VAR_INPUT
	bEnablePV		: BOOL; (* enable present value with priority x in priority array, FALSE = priority x disable *)
	bNullPV			: BOOL; (* clear priority entry *)
	fPV				: REAL; (* decimal number for priority x, when input bEnablePV is TRUE *)
END_VAR
VAR_IN_OUT
	Device			: FB_BACnet_Device;
END_VAR
VAR_OUTPUT
	bReady			: BOOL;
	fPresentValue	: REAL;
	bOverridden		: BOOL;
	bOutOfService	: BOOL;
	bFault			: BOOL;
	bInAlarm		: BOOL;
	bError			: BOOL;
	nErrorId		: UINT;
END_VAR
VAR
	_PresentValue AT%I*: REAL; 			(* ~(BACnet_PresentValue 			:		: )
								   			(BACnet_ObjectType 				: AO	: )	*)
    _PresentValue_Priority12 AT%Q*: DWORD;(* ~(BACnet_PresentValue_Priority12:		: )	*)
	_StatusFlags AT%I*: WORD; 			(* ~(BACnet_StatusFlags 			:		: )	*)
	_StatusFlagsBits : ST_BACnet_StatusFlags;
	_nUpdateCount : UDINT := 0;
END_VAR
(* update server device *)
IF (Device._nUpdateCount = _nUpdateCount) THEN
	Device();
END_IF
(* remind current number of update counter *)
_nUpdateCount := Device._nUpdateCount;

IF Device.bFirstCycle THEN
	(* first call of the server device since reboot/reset *)
	bReady := FALSE;
	_PresentValue_Priority12 := F_BACnet_RealNothing();

ELSIF (_StatusFlags < 4) THEN
	(* wrong mapping *)
	nErrorId := BACnet_ERR_WRONG_MAPPING;
	bReady := FALSE;

ELSIF Device.bOperational THEN
	(* ready state *)
	bReady := TRUE;
	nErrorId := BACnet_ERR_NO_ERROR;

	(* write into priority array *)
	_PresentValue_Priority12 := F_BACnet_RealPV(bEnablePV, bNullPV, fPV);

	(* present value *)
	fPresentValue := _PresentValue;

	(* build bit states *)
	_StatusFlagsBits := F_BACnet_StatusFlags(_StatusFlags);

	(* copy states to output *)
	bOverridden := _StatusFlagsBits.overridden;
	bOutOfService := _StatusFlagsBits.out_of_service;
	bFault := _StatusFlagsBits.fault;
	bInAlarm := _StatusFlagsBits.in_alarm;

ELSE
	(* server device not ready, reset local ready also *)
	bReady := FALSE;
	nErrorId := BACnet_ERR_OPERATIONAL;
END_IF
(* set error flag *)
bError := (nErrorId <> BACnet_ERR_NO_ERROR);
END_FUNCTION_BLOCK

(* POU FB_BACnet_AnalogOutput_ADS, ST *)
FUNCTION_BLOCK FB_BACnet_AnalogOutput_ADS
VAR_INPUT
	bEnablePV			: BOOL; (* enable PV write commands *)
	bNullPV				: BOOL; (* clear priority entry *)
	fPV					: REAL; (* decimal number for priority x, when input bEnablePV is TRUE and bNullPV is FALSE *)
	bManual				: BOOL; (* FALSE --> TRUE: write present_value immediately, FALSE: only write present_value on-change, TRUE: write present_value on-change and when device turns operational *)
	ePriority			: E_BACNETPRIORITY := BACNETPRIORITY_12;
END_VAR
VAR_IN_OUT
	Device				: FB_BACnet_Device;
END_VAR
VAR_OUTPUT
	bReady				: BOOL;
	bPvDone				: BOOL; (* present_value written over ADS *)
	fPresentValue		: REAL;
	bOverridden			: BOOL;
	bOutOfService		: BOOL;
	bFault				: BOOL;
	bInAlarm			: BOOL;
	tObjectID			: T_BACnet_ObjectIdentifier := 16#FFFFFFFF;
	bError				: BOOL;
	nErrorId			: UINT;
	nAdsErrorId			: UDINT;
END_VAR
VAR
	_PresentValue AT%I*: REAL; 			(* ~(BACnet_PresentValue 		:		: )
								   			(BACnet_ObjectType 			: AO	: )	*)
    _PresentValue_Ads : DWORD;
	_ObjectId AT%I*: DWORD;				(* ~(BACnet_ObjectIdentifier	:		: LINK) *)
	_StatusFlags AT%I*: WORD; 			(* ~(BACnet_StatusFlags 		:		: )	*)
	_StatusFlagsBits : ST_BACnet_StatusFlags;
	_nUpdateCount : UDINT := 0;
	_WriteProp : FB_BACnet_WriteProp;
	_rtrigManual : R_TRIG;
	_bNullPvOld : BOOL;
	_nObjType : E_BACNETOBJECTTYPE;
END_VAR
(* update server device *)
IF (Device._nUpdateCount = _nUpdateCount) THEN
	Device();
END_IF
(* remind current number of update counter *)
_nUpdateCount := Device._nUpdateCount;

(* trigger on manual flag *)
_rtrigManual(CLK:= bManual, Q=> );

(* decode object type *)
_nObjType := F_BACnet_GetObjType(_ObjectId);

IF Device.bFirstCycle THEN
	(* first call of the server device since reboot/reset *)
	bReady := FALSE;
	bPvDone := FALSE;

ELSIF _nObjType <> BACnetObjectType_AnalogOutput THEN
	(* wrong mapped object type *)
	nErrorId := BACnet_ERR_INVALID_OBJECTTYPE;
	bReady := FALSE;
	bPvDone := FALSE;

ELSIF (_StatusFlags < 4) THEN
	(* wrong mapping *)
	nErrorId := BACnet_ERR_WRONG_MAPPING;
	bReady := FALSE;
	bPvDone := FALSE;

ELSIF Device.bOperational THEN

	IF Device.stAdsConn.bValid THEN
		(* write present_value on manual trigger, on-change and on operational recover *)
		IF		bEnablePV
			AND	(		_rtrigManual.Q
					OR	(MEMCMP(pBuf1:=ADR(fPV), pBuf2:=ADR(_PresentValue_Ads), n:=SIZEOF(_PresentValue_Ads)) <> 0)
					OR	((NOT bReady) AND bManual)
					OR	(bNullPV <> _bNullPvOld)
				)
		THEN
			_WriteProp.bExecute := TRUE;
			bPvDone := FALSE;
			(* write depending on enable state *)
			_PresentValue_Ads := F_BACnet_RealPV(TRUE, bNullPV, fPV);
			(* remind null flag *)
			_bNullPvOld := bNullPV;
		END_IF

		(* ready state *)
		IF (nAdsErrorId = 0) THEN
			bReady := TRUE;
			nErrorId := BACnet_ERR_NO_ERROR;
		END_IF

	ELSE
		(* invalid ADS connection *)
		bReady := FALSE;
		nErrorId := BACnet_ERR_INVALID_ADS_CONN;
		bPvDone := FALSE;
	END_IF

	(* present value *)
	fPresentValue := _PresentValue;

	(* build bit states *)
	_StatusFlagsBits := F_BACnet_StatusFlags(_StatusFlags);

	(* copy states to output *)
	bOverridden := _StatusFlagsBits.overridden;
	bOutOfService := _StatusFlagsBits.out_of_service;
	bFault := _StatusFlagsBits.fault;
	bInAlarm := _StatusFlagsBits.in_alarm;
	tObjectID := _ObjectId;

ELSE
	(* server device not ready, reset local ready also *)
	bReady := FALSE;
	nErrorId := BACnet_ERR_OPERATIONAL;
	bPvDone := FALSE;
END_IF

(* call write property command *)
_WriteProp(
	BACnetDevicePort	:= Device.stAdsConn.nAmsPort,
	bExecute			:= ,
	sNetId				:= Device.stAdsConn.sAmsNetId,
	ObjectType			:= _nObjType,
	PropertyID			:= BACnetPropertyIdentifier_PresentValue,
	Priority			:= ePriority,
	DataType			:= BACnetDataType_Real,
	ObjectInstance		:= F_BACnet_GetObjInstance(_ObjectId),
	ptrValue			:= ADR(_PresentValue_Ads),
	nLenValue			:= SIZEOF(_PresentValue_Ads),
	bDone				=> ,
	bBusy				=> ,
	bError				=> ,
	nErrID				=> );

(* set done flag *)
IF _WriteProp.bExecute AND (NOT _WriteProp.bBusy) THEN
	(* check if command was finished with error *)
	IF _WriteProp.bError THEN
		bPvDone		:= FALSE;
		bReady		:= FALSE;
		nErrorId	:= BACnet_ERR_ADS_Write;
	ELSE
		(* successful written *)
		bPvDone		:= TRUE;
	END_IF
	nAdsErrorId := _WriteProp.nErrID;
	(* reset execution bit *)
	_WriteProp(bExecute := FALSE);
END_IF

(* set error flag *)
bError := (nErrorId <> BACnet_ERR_NO_ERROR) OR (nAdsErrorId <> 0);
END_FUNCTION_BLOCK

